LIN {X 0,Y 265.309,Z 598.013,A -85,B 0,C 180,E1 -22713.344,E2 -22713.344} C_VEL
LIN {X 0,Y 272.116,Z 583.48,A -85,B 0,C 180,E1 -22714.4,E2 -22714.4} C_VEL
LIN {X 0,Y 277.319,Z 569.981,A -85,B 0,C 180,E1 -22715.135,E2 -22715.135} C_VEL
LIN {X 0,Y 276.814,Z 571.467,A -85,B 0,C 180,E1 -22715.465,E2 -22715.465} C_VEL
LIN {X 0,Y 273.942,Z 579.172,A -85,B 0,C 180,E1 -22715.833,E2 -22715.833} C_VEL
LIN {X 0,Y 271.697,Z 584.628,A -85,B 0,C 180,E1 -22715.976,E2 -22715.976} C_VEL
LIN {X 0,Y 263.827,Z 600.629,A -85,B 0,C 180,E1 -22715.795,E2 -22715.795} C_VEL
LIN {X 0,Y 261.002,Z 605.716,A -85,B 0,C 180,E1 -22715.928,E2 -22715.928} C_VEL
LIN {X 0,Y 260.072,Z 607.334,A -85,B 0,C 180,E1 -22716.034,E2 -22716.034} C_VEL
LIN {X 0,Y 251.746,Z 620.764,A -85,B 0,C 180,E1 -22717.282,E2 -22717.282} C_VEL
LIN {X 0,Y 243.261,Z 632.852,A -85,B 0,C 180,E1 -22718.732,E2 -22718.732} C_VEL
LIN {X 0,Y 233.8,Z 644.794,A -85,B 0,C 180,E1 -22720.62,E2 -22720.62} C_VEL
LIN {X 0,Y 224.848,Z 655.062,A -85,B 0,C 180,E1 -22722.729,E2 -22722.729} C_VEL
LIN {X 0,Y 215.182,Z 665.04,A -85,B 0,C 180,E1 -22725.393,E2 -22725.393} C_VEL
LIN {X 0,Y 206.221,Z 673.491,A -85,B 0,C 180,E1 -22728.348,E2 -22728.348} C_VEL
LIN {X 0,Y 198.032,Z 680.601,A -85,B 0,C 180,E1 -22731.603,E2 -22731.603} C_VEL
LIN {X 0,Y 190.807,Z 686.435,A -85,B 0,C 180,E1 -22735.183,E2 -22735.183} C_VEL
LIN {X 0,Y 183.186,Z 692.152,A -85,B 0,C 180,E1 -22740.079,E2 -22740.079} C_VEL
LIN {X 0,Y 178.076,Z 695.522,A -85,B 0,C 180,E1 -22744.267,E2 -22744.267} C_VEL
LIN {X 0,Y 174.051,Z 697.841,A -85,B 0,C 180,E1 -22748.687,E2 -22748.687} C_VEL
LIN {X 0,Y 171.345,Z 699.174,A -85,B 0,C 180,E1 -22753.311,E2 -22753.311} C_VEL
LIN {X 0,Y 169.67,Z 699.443,A -85,B 0,C 180,E1 -22758.044,E2 -22758.044} C_VEL
LIN {X 0,Y 168.987,Z 698.624,A -85,B 0,C 180,E1 -22762.829,E2 -22762.829} C_VEL
LIN {X 0,Y 169.136,Z 696.706,A -85,B 0,C 180,E1 -22767.615,E2 -22767.615} C_VEL
LIN {X 0,Y 169.279,Z 695.29,A -85,B 0,C 180,E1 -22769.996,E2 -22769.996} C_VEL
LIN {X 0,Y 169.245,Z 692.646,A -85,B 0,C 180,E1 -22773.352,E2 -22773.352} C_VEL
LIN {X 0,Y 169.28,Z 688.807,A -85,B 0,C 180,E1 -22777.151,E2 -22777.151} C_VEL
LIN {X 0,Y 169.775,Z 682.485,A -85,B 0,C 180,E1 -22781.942,E2 -22781.942} C_VEL
LIN {X 0,Y 170.866,Z 675.519,A -85,B 0,C 180,E1 -22786.115,E2 -22786.115} C_VEL
LIN {X 0,Y 172.718,Z 666.779,A -85,B 0,C 180,E1 -22790.36,E2 -22790.36} C_VEL
LIN {X 0,Y 175.16,Z 656.817,A -85,B 0,C 180,E1 -22794.28,E2 -22794.28} C_VEL
LIN {X 0,Y 177.808,Z 646.284,A -85,B 0,C 180,E1 -22797.669,E2 -22797.669} C_VEL
LIN {X 0,Y 180.909,Z 634.538,A -85,B 0,C 180,E1 -22800.765,E2 -22800.765} C_VEL
LIN {X 0,Y 184.216,Z 621.341,A -85,B 0,C 180,E1 -22803.582,E2 -22803.582} C_VEL
LIN {X 0,Y 187.346,Z 607.954,A -85,B 0,C 180,E1 -22805.88,E2 -22805.88} C_VEL
LIN {X 0,Y 190.597,Z 592.477,A -85,B 0,C 180,E1 -22807.971,E2 -22807.971} C_VEL
LIN {X 0,Y 193.235,Z 577.622,A -85,B 0,C 180,E1 -22809.525,E2 -22809.525} C_VEL
LIN {X 0,Y 195.597,Z 561.354,A -85,B 0,C 180,E1 -22810.781,E2 -22810.781} C_VEL
LIN {X 0,Y 197.639,Z 540.646,A -85,B 0,C 180,E1 -22811.89,E2 -22811.89} C_VEL
LIN {X 0,Y 204.347,Z 466.811,A -85,B 0,C 180,E1 -22815.376,E2 -22815.376} C_VEL
LIN {X 0,Y 196.162,Z 445.438,A -85,B 0,C 180,E1 -22818.116,E2 -22818.116} C_VEL
LIN {X 0,Y 186.895,Z 423.814,A -85,B 0,C 180,E1 -22821.346,E2 -22821.346} C_VEL
LIN {X 0,Y 180.833,Z 410.824,A -85,B 0,C 180,E1 -22823.629,E2 -22823.629} C_VEL
LIN {X 0,Y 174.86,Z 400.671,A -85,B 0,C 180,E1 -22825.813,E2 -22825.813} C_VEL
LIN {X 0,Y 172.955,Z 397.334,A -85,B 0,C 180,E1 -22826.558,E2 -22826.558} C_VEL
LIN {X 0,Y 171.581,Z 394.658,A -85,B 0,C 180,E1 -22827.132,E2 -22827.132} C_VEL
LIN {X 0,Y 171.407,Z 393.76,A -85,B 0,C 180,E1 -22827.269,E2 -22827.269} C_VEL
LIN {X 0,Y 171.396,Z 393.759,A -85,B 0,C 180,E1 -22830.525,E2 -22830.525} C_VEL
LIN {X 0,Y 171.391,Z 393.755,A -85,B 0,C 180,E1 -22835.792,E2 -22835.792} C_VEL
LIN {X 0,Y 171.496,Z 393.731,A -85,B 0,C 180,E1 -22840.863,E2 -22840.863} C_VEL
LIN {X 0,Y 171.535,Z 393.744,A -85,B 0,C 180,E1 -22845.77,E2 -22845.77} C_VEL
LIN {X 0,Y 171.829,Z 393.686,A -85,B 0,C 180,E1 -22850.584,E2 -22850.584} C_VEL
LIN {X 0,Y 171.769,Z 393.713,A -85,B 0,C 180,E1 -22855.307,E2 -22855.307} C_VEL
LIN {X 0,Y 172.297,Z 393.65,A -85,B 0,C 180,E1 -22860.001,E2 -22860.001} C_VEL
LIN {X 0,Y 171.83,Z 393.704,A -85,B 0,C 180,E1 -22866.865,E2 -22866.865} C_VEL
LIN {X 0,Y 171.755,Z 393.708,A -85,B 0,C 180,E1 -22870.895,E2 -22870.895} C_VEL
LIN {X 0,Y 171.498,Z 393.739,A -85,B 0,C 180,E1 -22876.671,E2 -22876.671} C_VEL
LIN {X 0,Y 171.468,Z 393.746,A -85,B 0,C 180,E1 -22879.502,E2 -22879.502} C_VEL
LIN {X 0,Y 171.392,Z 393.749,A -85,B 0,C 180,E1 -22885.572,E2 -22885.572} C_VEL
LIN {X 0,Y 171.408,Z 393.757,A -85,B 0,C 180,E1 -22890.575,E2 -22890.575} C_VEL
LIN {X 0,Y 171.383,Z 393.751,A -85,B 0,C 180,E1 -22895.038,E2 -22895.038} C_VEL
LIN {X 0,Y 171.335,Z 393.766,A -85,B 0,C 180,E1 -22898.804,E2 -22898.804} C_VEL
LIN {X 0,Y 171.311,Z 393.764,A -85,B 0,C 180,E1 -22904.222,E2 -22904.222} C_VEL
LIN {X 0,Y 171.323,Z 393.764,A -85,B 0,C 180,E1 -22908.983,E2 -22908.983} C_VEL
LIN {X 0,Y 171.354,Z 393.757,A -85,B 0,C 180,E1 -22912.037,E2 -22912.037} C_VEL
LIN {X 0,Y 171.393,Z 393.76,A -85,B 0,C 180,E1 -22915.097,E2 -22915.097} C_VEL
LIN {X 0,Y 171.404,Z 393.757,A -85,B 0,C 180,E1 -22920.53,E2 -22920.53} C_VEL
LIN {X 0,Y 171.427,Z 393.749,A -85,B 0,C 180,E1 -22925.801,E2 -22925.801} C_VEL
LIN {X 0,Y 171.517,Z 393.743,A -85,B 0,C 180,E1 -22930.868,E2 -22930.868} C_VEL
LIN {X 0,Y 171.561,Z 393.709,A -85,B 0,C 180,E1 -22935.775,E2 -22935.775} C_VEL
LIN {X 0,Y 171.844,Z 393.704,A -85,B 0,C 180,E1 -22940.588,E2 -22940.588} C_VEL
LIN {X 0,Y 171.784,Z 393.691,A -85,B 0,C 180,E1 -22945.31,E2 -22945.31} C_VEL
LIN {X 0,Y 172.313,Z 393.647,A -85,B 0,C 180,E1 -22950.003,E2 -22950.003} C_VEL
LIN {X 0,Y 171.79,Z 393.709,A -85,B 0,C 180,E1 -22954.697,E2 -22954.697} C_VEL
LIN {X 0,Y 171.848,Z 393.694,A -85,B 0,C 180,E1 -22959.419,E2 -22959.419} C_VEL
LIN {X 0,Y 171.547,Z 393.732,A -85,B 0,C 180,E1 -22964.612,E2 -22964.612} C_VEL
LIN {X 0,Y 172.401,Z 396.369,A -85,B 0,C 180,E1 -22965.066,E2 -22965.066} C_VEL
LIN {X 0,Y 174.007,Z 398.835,A -85,B 0,C 180,E1 -22965.674,E2 -22965.674} C_VEL
LIN {X 0,Y 180.352,Z 409.954,A -85,B 0,C 180,E1 -22968.021,E2 -22968.021} C_VEL
LIN {X 0,Y 190.153,Z 428.23,A -85,B 0,C 180,E1 -22971.426,E2 -22971.426} C_VEL
LIN {X 0,Y 199.911,Z 448.405,A -85,B 0,C 180,E1 -22974.543,E2 -22974.543} C_VEL
LIN {X 0,Y 204.128,Z 458.127,A -85,B 0,C 180,E1 -22975.853,E2 -22975.853} C_VEL
LIN {X 0,Y 204.377,Z 459.114,A -85,B 0,C 180,E1 -22975.953,E2 -22975.953} C_VEL
LIN {X 0,Y 196.155,Z 546.834,A -85,B 0,C 180,E1 -22980.109,E2 -22980.109} C_VEL
LIN {X 0,Y 194.151,Z 562.34,A -85,B 0,C 180,E1 -22981.218,E2 -22981.218} C_VEL
LIN {X 0,Y 191.648,Z 578.197,A -85,B 0,C 180,E1 -22982.776,E2 -22982.776} C_VEL
LIN {X 0,Y 188.749,Z 592.941,A -85,B 0,C 180,E1 -22984.643,E2 -22984.643} C_VEL
LIN {X 0,Y 185.649,Z 607.015,A -85,B 0,C 180,E1 -22986.896,E2 -22986.896} C_VEL
LIN {X 0,Y 182.391,Z 620.466,A -85,B 0,C 180,E1 -22989.586,E2 -22989.586} C_VEL
LIN {X 0,Y 179.209,Z 632.933,A -85,B 0,C 180,E1 -22992.665,E2 -22992.665} C_VEL
LIN {X 0,Y 176.477,Z 643.375,A -85,B 0,C 180,E1 -22995.798,E2 -22995.798} C_VEL
LIN {X 0,Y 173.855,Z 654.051,A -85,B 0,C 180,E1 -22999.699,E2 -22999.699} C_VEL
LIN {X 0,Y 171.827,Z 662.83,A -85,B 0,C 180,E1 -23003.624,E2 -23003.624} C_VEL
LIN {X 0,Y 170.237,Z 671.195,A -85,B 0,C 180,E1 -23008.239,E2 -23008.239} C_VEL
LIN {X 0,Y 169.225,Z 677.779,A -85,B 0,C 180,E1 -23012.816,E2 -23012.816} C_VEL
LIN {X 0,Y 168.701,Z 681.95,A -85,B 0,C 180,E1 -23016.428,E2 -23016.428} C_VEL
LIN {X 0,Y 168.411,Z 685.58,A -85,B 0,C 180,E1 -23020.497,E2 -23020.497} C_VEL
LIN {X 0,Y 168.556,Z 687.74,A -85,B 0,C 180,E1 -23023.545,E2 -23023.545} C_VEL
LIN {X 0,Y 169.088,Z 689.995,A -85,B 0,C 180,E1 -23028.005,E2 -23028.005} C_VEL
LIN {X 0,Y 170.558,Z 691.354,A -85,B 0,C 180,E1 -23032.898,E2 -23032.898} C_VEL
LIN {X 0,Y 172.858,Z 691.573,A -85,B 0,C 180,E1 -23037.669,E2 -23037.669} C_VEL
LIN {X 0,Y 176.211,Z 690.641,A -85,B 0,C 180,E1 -23042.285,E2 -23042.285} C_VEL
LIN {X 0,Y 180.649,Z 688.635,A -85,B 0,C 180,E1 -23046.702,E2 -23046.702} C_VEL
LIN {X 0,Y 186.124,Z 685.561,A -85,B 0,C 180,E1 -23050.882,E2 -23050.882} C_VEL
LIN {X 0,Y 192.617,Z 681.32,A -85,B 0,C 180,E1 -23054.797,E2 -23054.797} C_VEL
LIN {X 0,Y 200.065,Z 675.862,A -85,B 0,C 180,E1 -23058.43,E2 -23058.43} C_VEL
LIN {X 0,Y 208.432,Z 669.025,A -85,B 0,C 180,E1 -23061.771,E2 -23061.771} C_VEL
LIN {X 0,Y 215.958,Z 662.271,A -85,B 0,C 180,E1 -23064.321,E2 -23064.321} C_VEL
LIN {X 0,Y 226.24,Z 652.056,A -85,B 0,C 180,E1 -23067.27,E2 -23067.27} C_VEL
LIN {X 0,Y 235.563,Z 641.593,A -85,B 0,C 180,E1 -23069.545,E2 -23069.545} C_VEL
LIN {X 0,Y 245.162,Z 629.6,A -85,B 0,C 180,E1 -23071.544,E2 -23071.544} C_VEL
LIN {X 0,Y 254.447,Z 616.272,A -85,B 0,C 180,E1 -23073.257,E2 -23073.257} C_VEL
LIN {X 0,Y 262.74,Z 602.507,A -85,B 0,C 180,E1 -23074.602,E2 -23074.602} C_VEL
LIN {X 0,Y 266.574,Z 595.227,A -85,B 0,C 180,E1 -23075.183,E2 -23075.183} C_VEL
LIN {X 0,Y 260.072,Z 607.334,A -85,B 0,C 180,E1 -23076.034,E2 -23076.034} C_VEL
LIN {X 0,Y 257.087,Z 612.343,A -85,B 0,C 180,E1 -23076.29,E2 -23076.29} C_VEL
LIN {X 0,Y 246.93,Z 626.983,A -85,B 0,C 180,E1 -23076.519,E2 -23076.519} C_VEL
LIN {X 0,Y 243.455,Z 631.505,A -85,B 0,C 180,E1 -23076.819,E2 -23076.819} C_VEL
LIN {X 0,Y 242.341,Z 632.921,A -85,B 0,C 180,E1 -23076.983,E2 -23076.983} C_VEL
LIN {X 0,Y 232.271,Z 645.047,A -85,B 0,C 180,E1 -23078.815,E2 -23078.815} C_VEL
LIN {X 0,Y 222.913,Z 655.104,A -85,B 0,C 180,E1 -23080.825,E2 -23080.825} C_VEL
LIN {X 0,Y 212.809,Z 664.976,A -85,B 0,C 180,E1 -23083.399,E2 -23083.399} C_VEL
LIN {X 0,Y 203.374,Z 673.297,A -85,B 0,C 180,E1 -23086.276,E2 -23086.276} C_VEL
LIN {X 0,Y 194.708,Z 680.311,A -85,B 0,C 180,E1 -23089.477,E2 -23089.477} C_VEL
LIN {X 0,Y 186.796,Z 686.155,A -85,B 0,C 180,E1 -23092.985,E2 -23092.985} C_VEL
LIN {X 0,Y 180.082,Z 690.756,A -85,B 0,C 180,E1 -23096.878,E2 -23096.878} C_VEL
LIN {X 0,Y 174.271,Z 694.399,A -85,B 0,C 180,E1 -23101.054,E2 -23101.054} C_VEL
LIN {X 0,Y 169.355,Z 697.037,A -85,B 0,C 180,E1 -23105.478,E2 -23105.478} C_VEL
LIN {X 0,Y 165.814,Z 698.599,A -85,B 0,C 180,E1 -23110.176,E2 -23110.176} C_VEL
LIN {X 0,Y 163.412,Z 699.182,A -85,B 0,C 180,E1 -23115.042,E2 -23115.042} C_VEL
LIN {X 0,Y 162.216,Z 698.761,A -85,B 0,C 180,E1 -23120.017,E2 -23120.017} C_VEL
LIN {X 0,Y 161.906,Z 697.196,A -85,B 0,C 180,E1 -23125.016,E2 -23125.016} C_VEL
LIN {X 0,Y 162.081,Z 695.984,A -85,B 0,C 180,E1 -23127.511,E2 -23127.511} C_VEL
LIN {X 0,Y 162.222,Z 694.453,A -85,B 0,C 180,E1 -23129.996,E2 -23129.996} C_VEL
LIN {X 0,Y 162.204,Z 691.823,A -85,B 0,C 180,E1 -23133.347,E2 -23133.347} C_VEL
LIN {X 0,Y 162.256,Z 687.647,A -85,B 0,C 180,E1 -23137.462,E2 -23137.462} C_VEL
LIN {X 0,Y 162.595,Z 682.924,A -85,B 0,C 180,E1 -23141.212,E2 -23141.212} C_VEL
LIN {X 0,Y 163.809,Z 675.047,A -85,B 0,C 180,E1 -23146.189,E2 -23146.189} C_VEL
LIN {X 0,Y 165.581,Z 666.653,A -85,B 0,C 180,E1 -23150.421,E2 -23150.421} C_VEL
LIN {X 0,Y 168.212,Z 656.197,A -85,B 0,C 180,E1 -23154.692,E2 -23154.692} C_VEL
LIN {X 0,Y 170.935,Z 645.589,A -85,B 0,C 180,E1 -23158.213,E2 -23158.213} C_VEL
LIN {X 0,Y 174.342,Z 632.997,A -85,B 0,C 180,E1 -23161.6,E2 -23161.6} C_VEL
LIN {X 0,Y 177.572,Z 620.489,A -85,B 0,C 180,E1 -23164.328,E2 -23164.328} C_VEL
LIN {X 0,Y 180.782,Z 607.031,A -85,B 0,C 180,E1 -23166.702,E2 -23166.702} C_VEL
LIN {X 0,Y 184.15,Z 591.506,A -85,B 0,C 180,E1 -23168.849,E2 -23168.849} C_VEL
LIN {X 0,Y 187.11,Z 575.285,A -85,B 0,C 180,E1 -23170.557,E2 -23170.557} C_VEL
LIN {X 0,Y 189.456,Z 559.085,A -85,B 0,C 180,E1 -23171.798,E2 -23171.798} C_VEL
LIN {X 0,Y 192.546,Z 526.859,A -85,B 0,C 180,E1 -23173.48,E2 -23173.48} C_VEL
LIN {X 0,Y 198.059,Z 468.566,A -85,B 0,C 180,E1 -23176.293,E2 -23176.293} C_VEL
LIN {X 0,Y 190.091,Z 447.695,A -85,B 0,C 180,E1 -23179.074,E2 -23179.074} C_VEL
LIN {X 0,Y 180.267,Z 424.517,A -85,B 0,C 180,E1 -23182.73,E2 -23182.73} C_VEL
LIN {X 0,Y 174.823,Z 413.322,A -85,B 0,C 180,E1 -23184.82,E2 -23184.82} C_VEL
LIN {X 0,Y 167.745,Z 401.33,A -85,B 0,C 180,E1 -23187.598,E2 -23187.598} C_VEL
LIN {X 0,Y 166.305,Z 398.723,A -85,B 0,C 180,E1 -23188.218,E2 -23188.218} C_VEL
LIN {X 0,Y 164.725,Z 396.211,A -85,B 0,C 180,E1 -23188.875,E2 -23188.875} C_VEL
LIN {X 0,Y 164.37,Z 394.637,A -85,B 0,C 180,E1 -23189.131,E2 -23189.131} C_VEL
LIN {X 0,Y 164.345,Z 394.626,A -85,B 0,C 180,E1 -23194.683,E2 -23194.683} C_VEL
LIN {X 0,Y 164.404,Z 394.617,A -85,B 0,C 180,E1 -23200.117,E2 -23200.117} C_VEL
LIN {X 0,Y 164.464,Z 394.625,A -85,B 0,C 180,E1 -23205.144,E2 -23205.144} C_VEL
LIN {X 0,Y 164.75,Z 394.565,A -85,B 0,C 180,E1 -23210.176,E2 -23210.176} C_VEL
LIN {X 0,Y 164.805,Z 394.576,A -85,B 0,C 180,E1 -23212.651,E2 -23212.651} C_VEL
LIN {X 0,Y 165.261,Z 394.526,A -85,B 0,C 180,E1 -23220.001,E2 -23220.001} C_VEL
LIN {X 0,Y 164.808,Z 394.581,A -85,B 0,C 180,E1 -23227.351,E2 -23227.351} C_VEL
LIN {X 0,Y 164.69,Z 394.588,A -85,B 0,C 180,E1 -23231.059,E2 -23231.059} C_VEL
LIN {X 0,Y 164.42,Z 394.618,A -85,B 0,C 180,E1 -23237.411,E2 -23237.411} C_VEL
LIN {X 0,Y 164.409,Z 394.628,A -85,B 0,C 180,E1 -23239.998,E2 -23239.998} C_VEL
LIN {X 0,Y 164.328,Z 394.628,A -85,B 0,C 180,E1 -23246.097,E2 -23246.097} C_VEL
LIN {X 0,Y 164.348,Z 394.637,A -85,B 0,C 180,E1 -23251.22,E2 -23251.22} C_VEL
LIN {X 0,Y 164.271,Z 394.644,A -85,B 0,C 180,E1 -23256.796,E2 -23256.796} C_VEL
LIN {X 0,Y 164.278,Z 394.643,A -85,B 0,C 180,E1 -23259.921,E2 -23259.921} C_VEL
LIN {X 0,Y 164.273,Z 394.635,A -85,B 0,C 180,E1 -23263.345,E2 -23263.345} C_VEL
LIN {X 0,Y 164.253,Z 394.648,A -85,B 0,C 180,E1 -23266.801,E2 -23266.801} C_VEL
LIN {X 0,Y 164.283,Z 394.633,A -85,B 0,C 180,E1 -23270.359,E2 -23270.359} C_VEL
LIN {X 0,Y 164.32,Z 394.641,A -85,B 0,C 180,E1 -23274.355,E2 -23274.355} C_VEL
LIN {X 0,Y 164.363,Z 394.626,A -85,B 0,C 180,E1 -23279.134,E2 -23279.134} C_VEL
LIN {X 0,Y 164.384,Z 394.628,A -85,B 0,C 180,E1 -23284.693,E2 -23284.693} C_VEL
LIN {X 0,Y 164.418,Z 394.628,A -85,B 0,C 180,E1 -23290.118,E2 -23290.118} C_VEL
LIN {X 0,Y 164.489,Z 394.587,A -85,B 0,C 180,E1 -23295.15,E2 -23295.15} C_VEL
LIN {X 0,Y 164.766,Z 394.587,A -85,B 0,C 180,E1 -23300.18,E2 -23300.18} C_VEL
LIN {X 0,Y 164.821,Z 394.571,A -85,B 0,C 180,E1 -23302.654,E2 -23302.654} C_VEL
LIN {X 0,Y 165.277,Z 394.523,A -85,B 0,C 180,E1 -23310.004,E2 -23310.004} C_VEL
LIN {X 0,Y 164.825,Z 394.578,A -85,B 0,C 180,E1 -23317.353,E2 -23317.353} C_VEL
LIN {X 0,Y 164.701,Z 394.593,A -85,B 0,C 180,E1 -23321.053,E2 -23321.053} C_VEL
LIN {X 0,Y 164.572,Z 394.731,A -85,B 0,C 180,E1 -23322.802,E2 -23322.802} C_VEL
LIN {X 0,Y 165.635,Z 397.611,A -85,B 0,C 180,E1 -23323.342,E2 -23323.342} C_VEL
LIN {X 0,Y 167.007,Z 399.607,A -85,B 0,C 180,E1 -23323.894,E2 -23323.894} C_VEL
LIN {X 0,Y 174.83,Z 413.347,A -85,B 0,C 180,E1 -23327.015,E2 -23327.015} C_VEL
LIN {X 0,Y 183.507,Z 429.583,A -85,B 0,C 180,E1 -23330.166,E2 -23330.166} C_VEL
LIN {X 0,Y 194.197,Z 451.552,A -85,B 0,C 180,E1 -23333.729,E2 -23333.729} C_VEL
LIN {X 0,Y 198.049,Z 460.512,A -85,B 0,C 180,E1 -23334.984,E2 -23334.984} C_VEL
LIN {X 0,Y 189.736,Z 546.86,A -85,B 0,C 180,E1 -23339.216,E2 -23339.216} C_VEL
LIN {X 0,Y 187.516,Z 563.366,A -85,B 0,C 180,E1 -23340.453,E2 -23340.453} C_VEL
LIN {X 0,Y 185.074,Z 578.251,A -85,B 0,C 180,E1 -23341.975,E2 -23341.975} C_VEL
LIN {X 0,Y 182.06,Z 593.007,A -85,B 0,C 180,E1 -23343.904,E2 -23343.904} C_VEL
LIN {X 0,Y 178.874,Z 607.033,A -85,B 0,C 180,E1 -23346.228,E2 -23346.228} C_VEL
LIN {X 0,Y 175.44,Z 620.856,A -85,B 0,C 180,E1 -23349.09,E2 -23349.09} C_VEL
LIN {X 0,Y 172.185,Z 633.307,A -85,B 0,C 180,E1 -23352.284,E2 -23352.284} C_VEL
LIN {X 0,Y 169.119,Z 644.742,A -85,B 0,C 180,E1 -23355.886,E2 -23355.886} C_VEL
LIN {X 0,Y 166.503,Z 655.245,A -85,B 0,C 180,E1 -23359.958,E2 -23359.958} C_VEL
LIN {X 0,Y 164.361,Z 664.416,A -85,B 0,C 180,E1 -23364.34,E2 -23364.34} C_VEL
LIN {X 0,Y 162.963,Z 671.977,A -85,B 0,C 180,E1 -23368.833,E2 -23368.833} C_VEL
LIN {X 0,Y 162.111,Z 677.559,A -85,B 0,C 180,E1 -23372.921,E2 -23372.921} C_VEL
LIN {X 0,Y 161.542,Z 682.055,A -85,B 0,C 180,E1 -23376.948,E2 -23376.948} C_VEL
LIN {X 0,Y 161.331,Z 685.518,A -85,B 0,C 180,E1 -23380.929,E2 -23380.929} C_VEL
LIN {X 0,Y 161.541,Z 688.197,A -85,B 0,C 180,E1 -23384.868,E2 -23384.868} C_VEL
LIN {X 0,Y 162.42,Z 690.538,A -85,B 0,C 180,E1 -23390.032,E2 -23390.032} C_VEL
LIN {X 0,Y 164.313,Z 691.706,A -85,B 0,C 180,E1 -23395.092,E2 -23395.092} C_VEL
LIN {X 0,Y 167.11,Z 691.771,A -85,B 0,C 180,E1 -23399.999,E2 -23399.999} C_VEL
LIN {X 0,Y 171.078,Z 690.75,A -85,B 0,C 180,E1 -23404.712,E2 -23404.712} C_VEL
LIN {X 0,Y 176.153,Z 688.62,A -85,B 0,C 180,E1 -23409.182,E2 -23409.182} C_VEL
LIN {X 0,Y 182.257,Z 685.406,A -85,B 0,C 180,E1 -23413.377,E2 -23413.377} C_VEL
LIN {X 0,Y 189.395,Z 681.103,A -85,B 0,C 180,E1 -23417.269,E2 -23417.269} C_VEL
LIN {X 0,Y 197.541,Z 675.543,A -85,B 0,C 180,E1 -23420.84,E2 -23420.84} C_VEL
LIN {X 0,Y 206.495,Z 668.649,A -85,B 0,C 180,E1 -23424.105,E2 -23424.105} C_VEL
LIN {X 0,Y 216.315,Z 660.244,A -85,B 0,C 180,E1 -23427.055,E2 -23427.055} C_VEL
LIN {X 0,Y 226.267,Z 650.649,A -85,B 0,C 180,E1 -23429.572,E2 -23429.572} C_VEL
LIN {X 0,Y 235.14,Z 641.085,A -85,B 0,C 180,E1 -23431.537,E2 -23431.537} C_VEL
LIN {X 0,Y 246.03,Z 627.844,A -85,B 0,C 180,E1 -23433.601,E2 -23433.601} C_VEL
LIN {X 0,Y 253.972,Z 616.755,A -85,B 0,C 180,E1 -23434.918,E2 -23434.918} C_VEL
LIN {X 0,Y 253.57,Z 617.352,A -85,B 0,C 180,E1 -23435.252,E2 -23435.252} C_VEL
LIN {X 0,Y 244.958,Z 629.559,A -85,B 0,C 180,E1 -23436.547,E2 -23436.547} C_VEL
LIN {X 0,Y 242.341,Z 632.921,A -85,B 0,C 180,E1 -23436.983,E2 -23436.983} C_VEL
LIN {X 0,Y 238.762,Z 637.308,A -85,B 0,C 180,E1 -23437.415,E2 -23437.415} C_VEL
LIN {X 0,Y 226.667,Z 650.086,A -85,B 0,C 180,E1 -23438.136,E2 -23438.136} C_VEL
LIN {X 0,Y 222.719,Z 653.943,A -85,B 0,C 180,E1 -23438.631,E2 -23438.631} C_VEL
LIN {X 0,Y 221.493,Z 655.128,A -85,B 0,C 180,E1 -23438.867,E2 -23438.867} C_VEL
LIN {X 0,Y 210.73,Z 664.996,A -85,B 0,C 180,E1 -23441.372,E2 -23441.372} C_VEL
LIN {X 0,Y 200.849,Z 673.215,A -85,B 0,C 180,E1 -23444.162,E2 -23444.162} C_VEL
LIN {X 0,Y 192.191,Z 679.736,A -85,B 0,C 180,E1 -23447.063,E2 -23447.063} C_VEL
LIN {X 0,Y 183.25,Z 685.885,A -85,B 0,C 180,E1 -23450.739,E2 -23450.739} C_VEL
LIN {X 0,Y 174.205,Z 691.497,A -85,B 0,C 180,E1 -23455.608,E2 -23455.608} C_VEL
LIN {X 0,Y 168.087,Z 694.815,A -85,B 0,C 180,E1 -23459.881,E2 -23459.881} C_VEL
LIN {X 0,Y 162.899,Z 697.166,A -85,B 0,C 180,E1 -23464.438,E2 -23464.438} C_VEL
LIN {X 0,Y 159.102,Z 698.562,A -85,B 0,C 180,E1 -23469.302,E2 -23469.302} C_VEL
LIN {X 0,Y 156.513,Z 698.895,A -85,B 0,C 180,E1 -23474.366,E2 -23474.366} C_VEL
LIN {X 0,Y 155.193,Z 698.241,A -85,B 0,C 180,E1 -23479.56,E2 -23479.56} C_VEL
LIN {X 0,Y 154.844,Z 696.538,A -85,B 0,C 180,E1 -23484.788,E2 -23484.788} C_VEL
LIN {X 0,Y 155.031,Z 695.248,A -85,B 0,C 180,E1 -23487.398,E2 -23487.398} C_VEL
LIN {X 0,Y 155.143,Z 692.648,A -85,B 0,C 180,E1 -23491.294,E2 -23491.294} C_VEL
LIN {X 0,Y 155.156,Z 689.213,A -85,B 0,C 180,E1 -23495.194,E2 -23495.194} C_VEL
LIN {X 0,Y 155.44,Z 683.237,A -85,B 0,C 180,E1 -23500.415,E2 -23500.415} C_VEL
LIN {X 0,Y 156.531,Z 675.556,A -85,B 0,C 180,E1 -23505.624,E2 -23505.624} C_VEL
LIN {X 0,Y 158.267,Z 667.228,A -85,B 0,C 180,E1 -23510.125,E2 -23510.125} C_VEL
LIN {X 0,Y 160.842,Z 657.16,A -85,B 0,C 180,E1 -23514.521,E2 -23514.521} C_VEL
LIN {X 0,Y 163.589,Z 646.763,A -85,B 0,C 180,E1 -23518.197,E2 -23518.197} C_VEL
LIN {X 0,Y 166.98,Z 634.461,A -85,B 0,C 180,E1 -23521.738,E2 -23521.738} C_VEL
LIN {X 0,Y 170.463,Z 621.478,A -85,B 0,C 180,E1 -23524.744,E2 -23524.744} C_VEL
LIN {X 0,Y 173.888,Z 607.625,A -85,B 0,C 180,E1 -23527.314,E2 -23527.314} C_VEL
LIN {X 0,Y 177.348,Z 592.313,A -85,B 0,C 180,E1 -23529.529,E2 -23529.529} C_VEL
LIN {X 0,Y 180.354,Z 576.352,A -85,B 0,C 180,E1 -23531.296,E2 -23531.296} C_VEL
LIN {X 0,Y 182.892,Z 559.849,A -85,B 0,C 180,E1 -23532.626,E2 -23532.626} C_VEL
LIN {X 0,Y 185.341,Z 535.37,A -85,B 0,C 180,E1 -23534.001,E2 -23534.001} C_VEL
LIN {X 0,Y 191.807,Z 470.279,A -85,B 0,C 180,E1 -23537.265,E2 -23537.265} C_VEL
LIN {X 0,Y 184.193,Z 450.466,A -85,B 0,C 180,E1 -23540.009,E2 -23540.009} C_VEL
LIN {X 0,Y 175.101,Z 428.62,A -85,B 0,C 180,E1 -23543.572,E2 -23543.572} C_VEL
LIN {X 0,Y 169.951,Z 417.871,A -85,B 0,C 180,E1 -23545.64,E2 -23545.64} C_VEL
LIN {X 0,Y 161.646,Z 403.553,A -85,B 0,C 180,E1 -23549.098,E2 -23549.098} C_VEL
LIN {X 0,Y 159.095,Z 399.449,A -85,B 0,C 180,E1 -23550.201,E2 -23550.201} C_VEL
LIN {X 0,Y 157.53,Z 396.844,A -85,B 0,C 180,E1 -23550.913,E2 -23550.913} C_VEL
LIN {X 0,Y 157.248,Z 395.523,A -85,B 0,C 180,E1 -23551.158,E2 -23551.158} C_VEL
LIN {X 0,Y 157.254,Z 395.519,A -85,B 0,C 180,E1 -23556.283,E2 -23556.283} C_VEL
LIN {X 0,Y 157.347,Z 395.498,A -85,B 0,C 180,E1 -23559.702,E2 -23559.702} C_VEL
LIN {X 0,Y 157.397,Z 395.506,A -85,B 0,C 180,E1 -23564.461,E2 -23564.461} C_VEL
LIN {X 0,Y 157.673,Z 395.444,A -85,B 0,C 180,E1 -23569.73,E2 -23569.73} C_VEL
LIN {X 0,Y 157.744,Z 395.452,A -85,B 0,C 180,E1 -23572.32,E2 -23572.32} C_VEL
LIN {X 0,Y 158.223,Z 395.403,A -85,B 0,C 180,E1 -23580.001,E2 -23580.001} C_VEL
LIN {X 0,Y 157.746,Z 395.46,A -85,B 0,C 180,E1 -23587.682,E2 -23587.682} C_VEL
LIN {X 0,Y 157.619,Z 395.469,A -85,B 0,C 180,E1 -23591.225,E2 -23591.225} C_VEL
LIN {X 0,Y 157.398,Z 395.5,A -85,B 0,C 180,E1 -23595.541,E2 -23595.541} C_VEL
LIN {X 0,Y 157.293,Z 395.516,A -85,B 0,C 180,E1 -23600.944,E2 -23600.944} C_VEL
LIN {X 0,Y 157.256,Z 395.511,A -85,B 0,C 180,E1 -23606.652,E2 -23606.652} C_VEL
LIN {X 0,Y 157.258,Z 395.513,A -85,B 0,C 180,E1 -23612.432,E2 -23612.432} C_VEL
LIN {X 0,Y 157.25,Z 395.518,A -85,B 0,C 180,E1 -23616.447,E2 -23616.447} C_VEL
LIN {X 0,Y 157.182,Z 395.516,A -85,B 0,C 180,E1 -23622.121,E2 -23622.121} C_VEL
LIN {X 0,Y 157.183,Z 395.528,A -85,B 0,C 180,E1 -23627.886,E2 -23627.886} C_VEL
LIN {X 0,Y 157.253,Z 395.52,A -85,B 0,C 180,E1 -23633.56,E2 -23633.56} C_VEL
LIN {X 0,Y 157.275,Z 395.508,A -85,B 0,C 180,E1 -23638.108,E2 -23638.108} C_VEL
LIN {X 0,Y 157.306,Z 395.514,A -85,B 0,C 180,E1 -23643.468,E2 -23643.468} C_VEL
LIN {X 0,Y 157.36,Z 395.509,A -85,B 0,C 180,E1 -23649.704,E2 -23649.704} C_VEL
LIN {X 0,Y 157.421,Z 395.467,A -85,B 0,C 180,E1 -23654.467,E2 -23654.467} C_VEL
LIN {X 0,Y 157.688,Z 395.468,A -85,B 0,C 180,E1 -23659.735,E2 -23659.735} C_VEL
LIN {X 0,Y 157.759,Z 395.453,A -85,B 0,C 180,E1 -23662.324,E2 -23662.324} C_VEL
LIN {X 0,Y 158.24,Z 395.4,A -85,B 0,C 180,E1 -23670.004,E2 -23670.004} C_VEL
LIN {X 0,Y 157.763,Z 395.455,A -85,B 0,C 180,E1 -23677.684,E2 -23677.684} C_VEL
LIN {X 0,Y 157.689,Z 395.584,A -85,B 0,C 180,E1 -23680.871,E2 -23680.871} C_VEL
LIN {X 0,Y 158.632,Z 398.311,A -85,B 0,C 180,E1 -23681.412,E2 -23681.412} C_VEL
LIN {X 0,Y 160.15,Z 400.763,A -85,B 0,C 180,E1 -23682.084,E2 -23682.084} C_VEL
LIN {X 0,Y 168.215,Z 414.667,A -85,B 0,C 180,E1 -23685.485,E2 -23685.485} C_VEL
LIN {X 0,Y 176.846,Z 430.82,A -85,B 0,C 180,E1 -23688.814,E2 -23688.814} C_VEL
LIN {X 0,Y 185.269,Z 447.999,A -85,B 0,C 180,E1 -23691.837,E2 -23691.837} C_VEL
LIN {X 0,Y 191.764,Z 462.177,A -85,B 0,C 180,E1 -23694.003,E2 -23694.003} C_VEL
LIN {X 0,Y 183.257,Z 547.205,A -85,B 0,C 180,E1 -23698.324,E2 -23698.324} C_VEL
LIN {X 0,Y 180.917,Z 564.042,A -85,B 0,C 180,E1 -23699.633,E2 -23699.633} C_VEL
LIN {X 0,Y 178.059,Z 580.471,A -85,B 0,C 180,E1 -23701.4,E2 -23701.4} C_VEL
LIN {X 0,Y 174.754,Z 596.036,A -85,B 0,C 180,E1 -23703.585,E2 -23703.585} C_VEL
LIN {X 0,Y 171.542,Z 609.511,A -85,B 0,C 180,E1 -23705.986,E2 -23705.986} C_VEL
LIN {X 0,Y 168.011,Z 623.108,A -85,B 0,C 180,E1 -23708.995,E2 -23708.995} C_VEL
LIN {X 0,Y 164.533,Z 635.938,A -85,B 0,C 180,E1 -23712.537,E2 -23712.537} C_VEL
LIN {X 0,Y 161.377,Z 647.629,A -85,B 0,C 180,E1 -23716.577,E2 -23716.577} C_VEL
LIN {X 0,Y 158.746,Z 657.704,A -85,B 0,C 180,E1 -23720.884,E2 -23720.884} C_VEL
LIN {X 0,Y 156.9,Z 665.915,A -85,B 0,C 180,E1 -23725.172,E2 -23725.172} C_VEL
LIN {X 0,Y 155.818,Z 671.947,A -85,B 0,C 180,E1 -23728.985,E2 -23728.985} C_VEL
LIN {X 0,Y 155.019,Z 677.331,A -85,B 0,C 180,E1 -23733.039,E2 -23733.039} C_VEL
LIN {X 0,Y 154.428,Z 681.878,A -85,B 0,C 180,E1 -23737.242,E2 -23737.242} C_VEL
LIN {X 0,Y 154.249,Z 685.419,A -85,B 0,C 180,E1 -23741.4,E2 -23741.4} C_VEL
LIN {X 0,Y 154.406,Z 687.327,A -85,B 0,C 180,E1 -23744.15,E2 -23744.15} C_VEL
LIN {X 0,Y 155.178,Z 690.14,A -85,B 0,C 180,E1 -23749.562,E2 -23749.562} C_VEL
LIN {X 0,Y 157.015,Z 691.703,A -85,B 0,C 180,E1 -23754.863,E2 -23754.863} C_VEL
LIN {X 0,Y 159.834,Z 692.14,A -85,B 0,C 180,E1 -23759.999,E2 -23759.999} C_VEL
LIN {X 0,Y 163.854,Z 691.532,A -85,B 0,C 180,E1 -23764.92,E2 -23764.92} C_VEL
LIN {X 0,Y 169.032,Z 689.884,A -85,B 0,C 180,E1 -23769.573,E2 -23769.573} C_VEL
LIN {X 0,Y 175.264,Z 687.126,A -85,B 0,C 180,E1 -23773.921,E2 -23773.921} C_VEL
LIN {X 0,Y 182.573,Z 683.259,A -85,B 0,C 180,E1 -23777.935,E2 -23777.935} C_VEL
LIN {X 0,Y 190.896,Z 678.27,A -85,B 0,C 180,E1 -23781.601,E2 -23781.601} C_VEL
LIN {X 0,Y 200.103,Z 671.985,A -85,B 0,C 180,E1 -23784.926,E2 -23784.926} C_VEL
LIN {X 0,Y 210.129,Z 664.269,A -85,B 0,C 180,E1 -23787.92,E2 -23787.92} C_VEL
LIN {X 0,Y 220.855,Z 654.973,A -85,B 0,C 180,E1 -23790.607,E2 -23790.607} C_VEL
LIN {X 0,Y 232.266,Z 643.68,A -85,B 0,C 180,E1 -23793,E2 -23793} C_VEL
LIN {X 0,Y 242.546,Z 632.074,A -85,B 0,C 180,E1 -23794.833,E2 -23794.833} C_VEL
LIN {X 0,Y 241.151,Z 633.824,A -85,B 0,C 180,E1 -23795.308,E2 -23795.308} C_VEL
LIN {X 0,Y 232.448,Z 643.864,A -85,B 0,C 180,E1 -23796.75,E2 -23796.75} C_VEL
LIN {X 0,Y 222.642,Z 653.995,A -85,B 0,C 180,E1 -23798.62,E2 -23798.62} C_VEL
LIN {X 0,Y 221.493,Z 655.128,A -85,B 0,C 180,E1 -23798.867,E2 -23798.867} C_VEL
LIN {X 0,Y 217.55,Z 658.797,A -85,B 0,C 180,E1 -23799.523,E2 -23799.523} C_VEL
LIN {X 0,Y 210.136,Z 664.816,A -85,B 0,C 180,E1 -23800.273,E2 -23800.273} C_VEL
LIN {X 0,Y 202.613,Z 670.365,A -85,B 0,C 180,E1 -23801.148,E2 -23801.148} C_VEL
LIN {X 0,Y 198.556,Z 673.248,A -85,B 0,C 180,E1 -23802.014,E2 -23802.014} C_VEL
LIN {X 0,Y 188.893,Z 680.038,A -85,B 0,C 180,E1 -23805.011,E2 -23805.011} C_VEL
LIN {X 0,Y 177.861,Z 686.91,A -85,B 0,C 180,E1 -23809.305,E2 -23809.305} C_VEL
LIN {X 0,Y 171.961,Z 690.236,A -85,B 0,C 180,E1 -23812.186,E2 -23812.186} C_VEL
LIN {X 0,Y 165.064,Z 693.784,A -85,B 0,C 180,E1 -23816.388,E2 -23816.388} C_VEL
LIN {X 0,Y 159.126,Z 696.389,A -85,B 0,C 180,E1 -23820.929,E2 -23820.929} C_VEL
LIN {X 0,Y 154.219,Z 697.97,A -85,B 0,C 180,E1 -23825.782,E2 -23825.782} C_VEL
LIN {X 0,Y 150.933,Z 698.624,A -85,B 0,C 180,E1 -23830.973,E2 -23830.973} C_VEL
LIN {X 0,Y 148.787,Z 698.278,A -85,B 0,C 180,E1 -23836.335,E2 -23836.335} C_VEL
LIN {X 0,Y 147.85,Z 696.875,A -85,B 0,C 180,E1 -23841.797,E2 -23841.797} C_VEL
LIN {X 0,Y 147.99,Z 694.389,A -85,B 0,C 180,E1 -23847.274,E2 -23847.274} C_VEL
LIN {X 0,Y 148.103,Z 691.648,A -85,B 0,C 180,E1 -23851.355,E2 -23851.355} C_VEL
LIN {X 0,Y 148.092,Z 688.103,A -85,B 0,C 180,E1 -23855.442,E2 -23855.442} C_VEL
LIN {X 0,Y 148.318,Z 683.55,A -85,B 0,C 180,E1 -23859.542,E2 -23859.542} C_VEL
LIN {X 0,Y 149.308,Z 676.013,A -85,B 0,C 180,E1 -23865,E2 -23865} C_VEL
LIN {X 0,Y 150.943,Z 667.827,A -85,B 0,C 180,E1 -23869.724,E2 -23869.724} C_VEL
LIN {X 0,Y 153.431,Z 657.931,A -85,B 0,C 180,E1 -23874.342,E2 -23874.342} C_VEL
LIN {X 0,Y 156.239,Z 647.804,A -85,B 0,C 180,E1 -23878.18,E2 -23878.18} C_VEL
LIN {X 0,Y 159.615,Z 635.785,A -85,B 0,C 180,E1 -23881.891,E2 -23881.891} C_VEL
LIN {X 0,Y 163.27,Z 622.707,A -85,B 0,C 180,E1 -23885.13,E2 -23885.13} C_VEL
LIN {X 0,Y 166.643,Z 609.727,A -85,B 0,C 180,E1 -23887.695,E2 -23887.695} C_VEL
LIN {X 0,Y 170.344,Z 594.08,A -85,B 0,C 180,E1 -23890.134,E2 -23890.134} C_VEL
LIN {X 0,Y 173.4,Z 578.732,A -85,B 0,C 180,E1 -23891.966,E2 -23891.966} C_VEL
LIN {X 0,Y 176.096,Z 562.237,A -85,B 0,C 180,E1 -23893.404,E2 -23893.404} C_VEL
LIN {X 0,Y 178.151,Z 543.789,A -85,B 0,C 180,E1 -23894.539,E2 -23894.539} C_VEL
LIN {X 0,Y 185.451,Z 471.895,A -85,B 0,C 180,E1 -23898.271,E2 -23898.271} C_VEL
LIN {X 0,Y 178.203,Z 452.791,A -85,B 0,C 180,E1 -23901.073,E2 -23901.073} C_VEL
LIN {X 0,Y 169.663,Z 432.156,A -85,B 0,C 180,E1 -23904.555,E2 -23904.555} C_VEL
LIN {X 0,Y 165.138,Z 422.44,A -85,B 0,C 180,E1 -23906.501,E2 -23906.501} C_VEL
LIN {X 0,Y 156.952,Z 408.221,A -85,B 0,C 180,E1 -23910.03,E2 -23910.03} C_VEL
LIN {X 0,Y 152.696,Z 401.107,A -85,B 0,C 180,E1 -23912.038,E2 -23912.038} C_VEL
LIN {X 0,Y 150.731,Z 398.245,A -85,B 0,C 180,E1 -23912.988,E2 -23912.988} C_VEL
LIN {X 0,Y 150.232,Z 396.385,A -85,B 0,C 180,E1 -23913.398,E2 -23913.398} C_VEL
LIN {X 0,Y 150.27,Z 396.383,A -85,B 0,C 180,E1 -23919.277,E2 -23919.277} C_VEL
LIN {X 0,Y 150.303,Z 396.385,A -85,B 0,C 180,E1 -23923.707,E2 -23923.707} C_VEL
LIN {X 0,Y 150.593,Z 396.325,A -85,B 0,C 180,E1 -23929.242,E2 -23929.242} C_VEL
LIN {X 0,Y 150.667,Z 396.331,A -85,B 0,C 180,E1 -23931.956,E2 -23931.956} C_VEL
LIN {X 0,Y 151.184,Z 396.28,A -85,B 0,C 180,E1 -23940.001,E2 -23940.001} C_VEL
LIN {X 0,Y 150.669,Z 396.339,A -85,B 0,C 180,E1 -23948.045,E2 -23948.045} C_VEL
LIN {X 0,Y 150.561,Z 396.348,A -85,B 0,C 180,E1 -23951.429,E2 -23951.429} C_VEL
LIN {X 0,Y 150.303,Z 396.379,A -85,B 0,C 180,E1 -23956.294,E2 -23956.294} C_VEL
LIN {X 0,Y 150.271,Z 396.391,A -85,B 0,C 180,E1 -23960.724,E2 -23960.724} C_VEL
LIN {X 0,Y 150.175,Z 396.395,A -85,B 0,C 180,E1 -23967.24,E2 -23967.24} C_VEL
LIN {X 0,Y 150.199,Z 396.392,A -85,B 0,C 180,E1 -23972.631,E2 -23972.631} C_VEL
LIN {X 0,Y 150.161,Z 396.403,A -85,B 0,C 180,E1 -23977.478,E2 -23977.478} C_VEL
LIN {X 0,Y 150.125,Z 396.397,A -85,B 0,C 180,E1 -23981.5,E2 -23981.5} C_VEL
LIN {X 0,Y 150.12,Z 396.407,A -85,B 0,C 180,E1 -23985.399,E2 -23985.399} C_VEL
LIN {X 0,Y 150.13,Z 396.402,A -85,B 0,C 180,E1 -23989.058,E2 -23989.058} C_VEL
LIN {X 0,Y 150.17,Z 396.4,A -85,B 0,C 180,E1 -23992.714,E2 -23992.714} C_VEL
LIN {X 0,Y 150.201,Z 396.392,A -85,B 0,C 180,E1 -23997.378,E2 -23997.378} C_VEL
LIN {X 0,Y 150.235,Z 396.396,A -85,B 0,C 180,E1 -24002.727,E2 -24002.727} C_VEL
LIN {X 0,Y 150.284,Z 396.392,A -85,B 0,C 180,E1 -24009.278,E2 -24009.278} C_VEL
LIN {X 0,Y 150.324,Z 396.353,A -85,B 0,C 180,E1 -24013.714,E2 -24013.714} C_VEL
LIN {X 0,Y 150.608,Z 396.347,A -85,B 0,C 180,E1 -24019.246,E2 -24019.246} C_VEL
LIN {X 0,Y 150.682,Z 396.335,A -85,B 0,C 180,E1 -24021.961,E2 -24021.961} C_VEL
LIN {X 0,Y 151.2,Z 396.277,A -85,B 0,C 180,E1 -24030.004,E2 -24030.004} C_VEL
LIN {X 0,Y 150.662,Z 396.333,A -85,B 0,C 180,E1 -24038.639,E2 -24038.639} C_VEL
LIN {X 0,Y 151.614,Z 399.128,A -85,B 0,C 180,E1 -24039.257,E2 -24039.257} C_VEL
LIN {X 0,Y 153.192,Z 401.28,A -85,B 0,C 180,E1 -24039.994,E2 -24039.994} C_VEL
LIN {X 0,Y 163.534,Z 419.434,A -85,B 0,C 180,E1 -24044.645,E2 -24044.645} C_VEL
LIN {X 0,Y 172.802,Z 437.165,A -85,B 0,C 180,E1 -24048.404,E2 -24048.404} C_VEL
LIN {X 0,Y 182.693,Z 457.87,A -85,B 0,C 180,E1 -24052.029,E2 -24052.029} C_VEL
LIN {X 0,Y 185.529,Z 464.326,A -85,B 0,C 180,E1 -24053.023,E2 -24053.023} C_VEL
LIN {X 0,Y 176.83,Z 547.578,A -85,B 0,C 180,E1 -24057.371,E2 -24057.371} C_VEL
LIN {X 0,Y 174.509,Z 563.727,A -85,B 0,C 180,E1 -24058.655,E2 -24058.655} C_VEL
LIN {X 0,Y 171.618,Z 579.943,A -85,B 0,C 180,E1 -24060.432,E2 -24060.432} C_VEL
LIN {X 0,Y 168.421,Z 594.718,A -85,B 0,C 180,E1 -24062.537,E2 -24062.537} C_VEL
LIN {X 0,Y 164.713,Z 609.855,A -85,B 0,C 180,E1 -24065.31,E2 -24065.31} C_VEL
LIN {X 0,Y 161.209,Z 622.853,A -85,B 0,C 180,E1 -24068.304,E2 -24068.304} C_VEL
LIN {X 0,Y 157.634,Z 635.683,A -85,B 0,C 180,E1 -24071.976,E2 -24071.976} C_VEL
LIN {X 0,Y 154.445,Z 647.136,A -85,B 0,C 180,E1 -24076.055,E2 -24076.055} C_VEL
LIN {X 0,Y 151.799,Z 657.094,A -85,B 0,C 180,E1 -24080.428,E2 -24080.428} C_VEL
LIN {X 0,Y 149.852,Z 665.47,A -85,B 0,C 180,E1 -24084.933,E2 -24084.933} C_VEL
LIN {X 0,Y 148.465,Z 673.387,A -85,B 0,C 180,E1 -24090.194,E2 -24090.194} C_VEL
LIN {X 0,Y 147.651,Z 678.798,A -85,B 0,C 180,E1 -24094.747,E2 -24094.747} C_VEL
LIN {X 0,Y 147.18,Z 684.148,A -85,B 0,C 180,E1 -24100.472,E2 -24100.472} C_VEL
LIN {X 0,Y 147.297,Z 686.298,A -85,B 0,C 180,E1 -24103.364,E2 -24103.364} C_VEL
LIN {X 0,Y 147.942,Z 689.514,A -85,B 0,C 180,E1 -24109.045,E2 -24109.045} C_VEL
LIN {X 0,Y 149.722,Z 691.521,A -85,B 0,C 180,E1 -24114.612,E2 -24114.612} C_VEL
LIN {X 0,Y 152.547,Z 692.404,A -85,B 0,C 180,E1 -24119.999,E2 -24119.999} C_VEL
LIN {X 0,Y 156.592,Z 692.177,A -85,B 0,C 180,E1 -24125.149,E2 -24125.149} C_VEL
LIN {X 0,Y 161.878,Z 690.936,A -85,B 0,C 180,E1 -24130,E2 -24130} C_VEL
LIN {X 0,Y 168.285,Z 688.688,A -85,B 0,C 180,E1 -24134.511,E2 -24134.511} C_VEL
LIN {X 0,Y 177.793,Z 684.313,A -85,B 0,C 180,E1 -24139.633,E2 -24139.633} C_VEL
LIN {X 0,Y 186.582,Z 679.523,A -85,B 0,C 180,E1 -24143.297,E2 -24143.297} C_VEL
LIN {X 0,Y 196.835,Z 673.098,A -85,B 0,C 180,E1 -24146.789,E2 -24146.789} C_VEL
LIN {X 0,Y 207.993,Z 665.11,A -85,B 0,C 180,E1 -24149.893,E2 -24149.893} C_VEL
LIN {X 0,Y 219.256,Z 655.891,A -85,B 0,C 180,E1 -24152.473,E2 -24152.473} C_VEL
LIN {X 0,Y 228.971,Z 646.928,A -85,B 0,C 180,E1 -24154.379,E2 -24154.379} C_VEL
LIN {X 0,Y 230.891,Z 645.019,A -85,B 0,C 180,E1 -24154.727,E2 -24154.727} C_VEL
LIN {X 0,Y 231.478,Z 644.414,A -85,B 0,C 180,E1 -24154.936,E2 -24154.936} C_VEL
LIN {X 0,Y 221.328,Z 654.402,A -85,B 0,C 180,E1 -24156.696,E2 -24156.696} C_VEL
LIN {X 0,Y 208.977,Z 665.181,A -85,B 0,C 180,E1 -24159.327,E2 -24159.327} C_VEL
LIN {X 0,Y 198.556,Z 673.248,A -85,B 0,C 180,E1 -24162.014,E2 -24162.014} C_VEL
LIN {X 0,Y 194.458,Z 676.088,A -85,B 0,C 180,E1 -24162.954,E2 -24162.954} C_VEL
LIN {X 0,Y 186.668,Z 680.646,A -85,B 0,C 180,E1 -24164.202,E2 -24164.202} C_VEL
LIN {X 0,Y 178.871,Z 684.694,A -85,B 0,C 180,E1 -24165.615,E2 -24165.615} C_VEL
LIN {X 0,Y 174.839,Z 686.73,A -85,B 0,C 180,E1 -24166.827,E2 -24166.827} C_VEL
LIN {X 0,Y 166.434,Z 691.029,A -85,B 0,C 180,E1 -24170.694,E2 -24170.694} C_VEL
LIN {X 0,Y 159.204,Z 694.259,A -85,B 0,C 180,E1 -24174.975,E2 -24174.975} C_VEL
LIN {X 0,Y 152.942,Z 696.564,A -85,B 0,C 180,E1 -24179.633,E2 -24179.633} C_VEL
LIN {X 0,Y 147.664,Z 697.971,A -85,B 0,C 180,E1 -24184.727,E2 -24184.727} C_VEL
LIN {X 0,Y 144.188,Z 698.331,A -85,B 0,C 180,E1 -24190.046,E2 -24190.046} C_VEL
LIN {X 0,Y 141.874,Z 697.775,A -85,B 0,C 180,E1 -24195.655,E2 -24195.655} C_VEL
LIN {X 0,Y 140.837,Z 696.197,A -85,B 0,C 180,E1 -24201.386,E2 -24201.386} C_VEL
LIN {X 0,Y 140.945,Z 693.494,A -85,B 0,C 180,E1 -24207.138,E2 -24207.138} C_VEL
LIN {X 0,Y 141.065,Z 690.623,A -85,B 0,C 180,E1 -24211.423,E2 -24211.423} C_VEL
LIN {X 0,Y 141.074,Z 686.809,A -85,B 0,C 180,E1 -24215.714,E2 -24215.714} C_VEL
LIN {X 0,Y 141.316,Z 682.136,A -85,B 0,C 180,E1 -24220.02,E2 -24220.02} C_VEL
LIN {X 0,Y 142.402,Z 674.354,A -85,B 0,C 180,E1 -24225.746,E2 -24225.746} C_VEL
LIN {X 0,Y 144.226,Z 665.863,A -85,B 0,C 180,E1 -24230.684,E2 -24230.684} C_VEL
LIN {X 0,Y 146.988,Z 655.617,A -85,B 0,C 180,E1 -24235.483,E2 -24235.483} C_VEL
LIN {X 0,Y 149.942,Z 645.079,A -85,B 0,C 180,E1 -24239.477,E2 -24239.477} C_VEL
LIN {X 0,Y 153.596,Z 632.567,A -85,B 0,C 180,E1 -24243.299,E2 -24243.299} C_VEL
LIN {X 0,Y 157.187,Z 619.868,A -85,B 0,C 180,E1 -24246.41,E2 -24246.41} C_VEL
LIN {X 0,Y 161.004,Z 605.178,A -85,B 0,C 180,E1 -24249.262,E2 -24249.262} C_VEL
LIN {X 0,Y 164.687,Z 589.519,A -85,B 0,C 180,E1 -24251.61,E2 -24251.61} C_VEL
LIN {X 0,Y 167.652,Z 574.393,A -85,B 0,C 180,E1 -24253.344,E2 -24253.344} C_VEL
LIN {X 0,Y 170.314,Z 557.801,A -85,B 0,C 180,E1 -24254.729,E2 -24254.729} C_VEL
LIN {X 0,Y 175.273,Z 511.209,A -85,B 0,C 180,E1 -24257.347,E2 -24257.347} C_VEL
LIN {X 0,Y 179.228,Z 473.675,A -85,B 0,C 180,E1 -24259.326,E2 -24259.326} C_VEL
LIN {X 0,Y 172.484,Z 455.829,A -85,B 0,C 180,E1 -24262.048,E2 -24262.048} C_VEL
LIN {X 0,Y 164.249,Z 435.52,A -85,B 0,C 180,E1 -24265.626,E2 -24265.626} C_VEL
LIN {X 0,Y 159.955,Z 426.407,A -85,B 0,C 180,E1 -24267.542,E2 -24267.542} C_VEL
LIN {X 0,Y 152.407,Z 413.122,A -85,B 0,C 180,E1 -24270.959,E2 -24270.959} C_VEL
LIN {X 0,Y 147.477,Z 405.104,A -85,B 0,C 180,E1 -24273.4,E2 -24273.4} C_VEL
LIN {X 0,Y 145.205,Z 401.446,A -85,B 0,C 180,E1 -24274.562,E2 -24274.562} C_VEL
LIN {X 0,Y 143.569,Z 399.016,A -85,B 0,C 180,E1 -24275.413,E2 -24275.413} C_VEL
LIN {X 0,Y 143.101,Z 397.276,A -85,B 0,C 180,E1 -24275.81,E2 -24275.81} C_VEL
LIN {X 0,Y 143.234,Z 397.253,A -85,B 0,C 180,E1 -24279.913,E2 -24279.913} C_VEL
LIN {X 0,Y 143.294,Z 397.261,A -85,B 0,C 180,E1 -24285.805,E2 -24285.805} C_VEL
LIN {X 0,Y 143.519,Z 397.207,A -85,B 0,C 180,E1 -24288.705,E2 -24288.705} C_VEL
LIN {X 0,Y 143.593,Z 397.207,A -85,B 0,C 180,E1 -24291.557,E2 -24291.557} C_VEL
LIN {X 0,Y 144.142,Z 397.157,A -85,B 0,C 180,E1 -24300.001,E2 -24300.001} C_VEL
LIN {X 0,Y 143.595,Z 397.219,A -85,B 0,C 180,E1 -24308.444,E2 -24308.444} C_VEL
LIN {X 0,Y 143.486,Z 397.23,A -85,B 0,C 180,E1 -24311.616,E2 -24311.616} C_VEL
LIN {X 0,Y 143.242,Z 397.255,A -85,B 0,C 180,E1 -24317.121,E2 -24317.121} C_VEL
LIN {X 0,Y 143.208,Z 397.271,A -85,B 0,C 180,E1 -24321.196,E2 -24321.196} C_VEL
LIN {X 0,Y 143.132,Z 397.275,A -85,B 0,C 180,E1 -24327.903,E2 -24327.903} C_VEL
LIN {X 0,Y 143.129,Z 397.267,A -85,B 0,C 180,E1 -24333.419,E2 -24333.419} C_VEL
LIN {X 0,Y 143.044,Z 397.288,A -85,B 0,C 180,E1 -24339.697,E2 -24339.697} C_VEL
LIN {X 0,Y 143.026,Z 397.281,A -85,B 0,C 180,E1 -24343.468,E2 -24343.468} C_VEL
LIN {X 0,Y 143.031,Z 397.293,A -85,B 0,C 180,E1 -24347.482,E2 -24347.482} C_VEL
LIN {X 0,Y 143.065,Z 397.277,A -85,B 0,C 180,E1 -24351.814,E2 -24351.814} C_VEL
LIN {X 0,Y 143.168,Z 397.267,A -85,B 0,C 180,E1 -24357.323,E2 -24357.323} C_VEL
LIN {X 0,Y 143.179,Z 397.276,A -85,B 0,C 180,E1 -24362.074,E2 -24362.074} C_VEL
LIN {X 0,Y 143.225,Z 397.27,A -85,B 0,C 180,E1 -24368.803,E2 -24368.803} C_VEL
LIN {X 0,Y 143.261,Z 397.239,A -85,B 0,C 180,E1 -24372.886,E2 -24372.886} C_VEL
LIN {X 0,Y 143.535,Z 397.225,A -85,B 0,C 180,E1 -24378.71,E2 -24378.71} C_VEL
LIN {X 0,Y 143.608,Z 397.218,A -85,B 0,C 180,E1 -24381.562,E2 -24381.562} C_VEL
LIN {X 0,Y 144.159,Z 397.154,A -85,B 0,C 180,E1 -24390.004,E2 -24390.004} C_VEL
LIN {X 0,Y 143.59,Z 397.229,A -85,B 0,C 180,E1 -24396.239,E2 -24396.239} C_VEL
LIN {X 0,Y 144.653,Z 400.163,A -85,B 0,C 180,E1 -24396.981,E2 -24396.981} C_VEL
LIN {X 0,Y 146.27,Z 402.243,A -85,B 0,C 180,E1 -24397.771,E2 -24397.771} C_VEL
LIN {X 0,Y 150.964,Z 410.344,A -85,B 0,C 180,E1 -24400.155,E2 -24400.155} C_VEL
LIN {X 0,Y 158.594,Z 423.808,A -85,B 0,C 180,E1 -24403.709,E2 -24403.709} C_VEL
LIN {X 0,Y 166.573,Z 439.133,A -85,B 0,C 180,E1 -24407.094,E2 -24407.094} C_VEL
LIN {X 0,Y 176.794,Z 460.559,A -85,B 0,C 180,E1 -24411.027,E2 -24411.027} C_VEL
LIN {X 0,Y 179.284,Z 466.471,A -85,B 0,C 180,E1 -24411.969,E2 -24411.969} C_VEL
LIN {X 0,Y 170.521,Z 547.124,A -85,B 0,C 180,E1 -24416.308,E2 -24416.308} C_VEL
LIN {X 0,Y 168.04,Z 563.853,A -85,B 0,C 180,E1 -24417.683,E2 -24417.683} C_VEL
LIN {X 0,Y 165.05,Z 579.966,A -85,B 0,C 180,E1 -24419.51,E2 -24419.51} C_VEL
LIN {X 0,Y 161.676,Z 595.019,A -85,B 0,C 180,E1 -24421.739,E2 -24421.739} C_VEL
LIN {X 0,Y 157.896,Z 609.954,A -85,B 0,C 180,E1 -24424.57,E2 -24424.57} C_VEL
LIN {X 0,Y 154.305,Z 622.987,A -85,B 0,C 180,E1 -24427.686,E2 -24427.686} C_VEL
LIN {X 0,Y 151.004,Z 634.508,A -85,B 0,C 180,E1 -24431.086,E2 -24431.086} C_VEL
LIN {X 0,Y 147.677,Z 645.997,A -85,B 0,C 180,E1 -24435.247,E2 -24435.247} C_VEL
LIN {X 0,Y 144.815,Z 656.534,A -85,B 0,C 180,E1 -24439.98,E2 -24439.98} C_VEL
LIN {X 0,Y 142.815,Z 664.925,A -85,B 0,C 180,E1 -24444.673,E2 -24444.673} C_VEL
LIN {X 0,Y 141.691,Z 670.943,A -85,B 0,C 180,E1 -24448.705,E2 -24448.705} C_VEL
LIN {X 0,Y 140.7,Z 677.519,A -85,B 0,C 180,E1 -24454.049,E2 -24454.049} C_VEL
LIN {X 0,Y 140.153,Z 682.751,A -85,B 0,C 180,E1 -24459.45,E2 -24459.45} C_VEL
LIN {X 0,Y 140.164,Z 685.131,A -85,B 0,C 180,E1 -24462.491,E2 -24462.491} C_VEL
LIN {X 0,Y 140.707,Z 688.756,A -85,B 0,C 180,E1 -24468.474,E2 -24468.474} C_VEL
LIN {X 0,Y 142.441,Z 691.169,A -85,B 0,C 180,E1 -24474.336,E2 -24474.336} C_VEL
LIN {X 0,Y 145.25,Z 692.454,A -85,B 0,C 180,E1 -24479.999,E2 -24479.999} C_VEL
LIN {X 0,Y 149.338,Z 692.698,A -85,B 0,C 180,E1 -24485.4,E2 -24485.4} C_VEL
LIN {X 0,Y 154.749,Z 691.855,A -85,B 0,C 180,E1 -24490.466,E2 -24490.466} C_VEL
LIN {X 0,Y 161.288,Z 690.022,A -85,B 0,C 180,E1 -24495.155,E2 -24495.155} C_VEL
LIN {X 0,Y 168.967,Z 687.191,A -85,B 0,C 180,E1 -24499.435,E2 -24499.435} C_VEL
LIN {X 0,Y 177.692,Z 683.197,A -85,B 0,C 180,E1 -24503.298,E2 -24503.298} C_VEL
LIN {X 0,Y 187.371,Z 678.032,A -85,B 0,C 180,E1 -24506.75,E2 -24506.75} C_VEL
LIN {X 0,Y 197.794,Z 671.69,A -85,B 0,C 180,E1 -24509.831,E2 -24509.831} C_VEL
LIN {X 0,Y 210.47,Z 662.782,A -85,B 0,C 180,E1 -24512.862,E2 -24512.862} C_VEL
LIN {X 0,Y 218.841,Z 656.174,A -85,B 0,C 180,E1 -24514.542,E2 -24514.542} C_VEL
LIN {X 0,Y 217.634,Z 657.226,A -85,B 0,C 180,E1 -24515.255,E2 -24515.255} C_VEL
LIN {X 0,Y 206.129,Z 666.543,A -85,B 0,C 180,E1 -24517.556,E2 -24517.556} C_VEL
LIN {X 0,Y 194.102,Z 675.155,A -85,B 0,C 180,E1 -24520.5,E2 -24520.5} C_VEL
LIN {X 0,Y 184.054,Z 681.511,A -85,B 0,C 180,E1 -24523.485,E2 -24523.485} C_VEL
LIN {X 0,Y 174.839,Z 686.73,A -85,B 0,C 180,E1 -24526.827,E2 -24526.827} C_VEL
LIN {X 0,Y 170.864,Z 688.645,A -85,B 0,C 180,E1 -24528.139,E2 -24528.139} C_VEL
LIN {X 0,Y 163.294,Z 691.549,A -85,B 0,C 180,E1 -24530.1,E2 -24530.1} C_VEL
LIN {X 0,Y 157.352,Z 693.481,A -85,B 0,C 180,E1 -24531.824,E2 -24531.824} C_VEL
LIN {X 0,Y 153.57,Z 694.674,A -85,B 0,C 180,E1 -24533.423,E2 -24533.423} C_VEL
LIN {X 0,Y 152.542,Z 694.989,A -85,B 0,C 180,E1 -24534.034,E2 -24534.034} C_VEL
LIN {X 0,Y 146.832,Z 696.73,A -85,B 0,C 180,E1 -24538.226,E2 -24538.226} C_VEL
LIN {X 0,Y 140.962,Z 697.866,A -85,B 0,C 180,E1 -24543.821,E2 -24543.821} C_VEL
LIN {X 0,Y 137.475,Z 698.032,A -85,B 0,C 180,E1 -24549.027,E2 -24549.027} C_VEL
LIN {X 0,Y 134.989,Z 697.207,A -85,B 0,C 180,E1 -24554.907,E2 -24554.907} C_VEL
LIN {X 0,Y 133.841,Z 695.418,A -85,B 0,C 180,E1 -24560.932,E2 -24560.932} C_VEL
LIN {X 0,Y 133.906,Z 692.554,A -85,B 0,C 180,E1 -24566.987,E2 -24566.987} C_VEL
LIN {X 0,Y 134.048,Z 689.484,A -85,B 0,C 180,E1 -24571.498,E2 -24571.498} C_VEL
LIN {X 0,Y 134.036,Z 685.505,A -85,B 0,C 180,E1 -24576.015,E2 -24576.015} C_VEL
LIN {X 0,Y 134.338,Z 680.582,A -85,B 0,C 180,E1 -24580.546,E2 -24580.546} C_VEL
LIN {X 0,Y 135.351,Z 673.589,A -85,B 0,C 180,E1 -24585.814,E2 -24585.814} C_VEL
LIN {X 0,Y 137.242,Z 665.068,A -85,B 0,C 180,E1 -24591.001,E2 -24591.001} C_VEL
LIN {X 0,Y 140.094,Z 654.743,A -85,B 0,C 180,E1 -24596.039,E2 -24596.039} C_VEL
LIN {X 0,Y 143.138,Z 644.138,A -85,B 0,C 180,E1 -24600.211,E2 -24600.211} C_VEL
LIN {X 0,Y 146.974,Z 631.492,A -85,B 0,C 180,E1 -24604.179,E2 -24604.179} C_VEL
LIN {X 0,Y 150.601,Z 618.917,A -85,B 0,C 180,E1 -24607.343,E2 -24607.343} C_VEL
LIN {X 0,Y 154.223,Z 605.402,A -85,B 0,C 180,E1 -24610.061,E2 -24610.061} C_VEL
LIN {X 0,Y 158.002,Z 589.842,A -85,B 0,C 180,E1 -24612.491,E2 -24612.491} C_VEL
LIN {X 0,Y 161.3,Z 573.591,A -85,B 0,C 180,E1 -24614.41,E2 -24614.41} C_VEL
LIN {X 0,Y 163.931,Z 557.525,A -85,B 0,C 180,E1 -24615.782,E2 -24615.782} C_VEL
LIN {X 0,Y 169.929,Z 502.98,A -85,B 0,C 180,E1 -24618.949,E2 -24618.949} C_VEL
LIN {X 0,Y 173.014,Z 475.397,A -85,B 0,C 180,E1 -24620.444,E2 -24620.444} C_VEL
LIN {X 0,Y 165.347,Z 455.04,A -85,B 0,C 180,E1 -24623.714,E2 -24623.714} C_VEL
LIN {X 0,Y 157.829,Z 436.727,A -85,B 0,C 180,E1 -24627.198,E2 -24627.198} C_VEL
LIN {X 0,Y 154.697,Z 430.169,A -85,B 0,C 180,E1 -24628.654,E2 -24628.654} C_VEL
LIN {X 0,Y 147.672,Z 417.613,A -85,B 0,C 180,E1 -24632.065,E2 -24632.065} C_VEL
LIN {X 0,Y 141.008,Z 406.687,A -85,B 0,C 180,E1 -24635.525,E2 -24635.525} C_VEL
LIN {X 0,Y 138.945,Z 403.395,A -85,B 0,C 180,E1 -24636.695,E2 -24636.695} C_VEL
LIN {X 0,Y 136.68,Z 400.238,A -85,B 0,C 180,E1 -24637.992,E2 -24637.992} C_VEL
LIN {X 0,Y 136.145,Z 398.148,A -85,B 0,C 180,E1 -24638.562,E2 -24638.562} C_VEL
LIN {X 0,Y 136.212,Z 398.145,A -85,B 0,C 180,E1 -24645.051,E2 -24645.051} C_VEL
LIN {X 0,Y 136.413,Z 398.094,A -85,B 0,C 180,E1 -24648.178,E2 -24648.178} C_VEL
LIN {X 0,Y 136.522,Z 398.082,A -85,B 0,C 180,E1 -24651.117,E2 -24651.117} C_VEL
LIN {X 0,Y 137.099,Z 398.034,A -85,B 0,C 180,E1 -24660.001,E2 -24660.001} C_VEL
LIN {X 0,Y 136.524,Z 398.097,A -85,B 0,C 180,E1 -24668.885,E2 -24668.885} C_VEL
LIN {X 0,Y 136.402,Z 398.113,A -85,B 0,C 180,E1 -24671.895,E2 -24671.895} C_VEL
LIN {X 0,Y 136.154,Z 398.137,A -85,B 0,C 180,E1 -24678.043,E2 -24678.043} C_VEL
LIN {X 0,Y 136.133,Z 398.153,A -85,B 0,C 180,E1 -24681.692,E2 -24681.692} C_VEL
LIN {X 0,Y 136.052,Z 398.161,A -85,B 0,C 180,E1 -24688.589,E2 -24688.589} C_VEL
LIN {X 0,Y 136.031,Z 398.15,A -85,B 0,C 180,E1 -24694.634,E2 -24694.634} C_VEL
LIN {X 0,Y 136.016,Z 398.166,A -85,B 0,C 180,E1 -24699.198,E2 -24699.198} C_VEL
LIN {X 0,Y 135.971,Z 398.16,A -85,B 0,C 180,E1 -24703.652,E2 -24703.652} C_VEL
LIN {X 0,Y 135.975,Z 398.17,A -85,B 0,C 180,E1 -24707.792,E2 -24707.792} C_VEL
LIN {X 0,Y 136.014,Z 398.154,A -85,B 0,C 180,E1 -24711.686,E2 -24711.686} C_VEL
LIN {X 0,Y 136.047,Z 398.162,A -85,B 0,C 180,E1 -24715.747,E2 -24715.747} C_VEL
LIN {X 0,Y 136.135,Z 398.153,A -85,B 0,C 180,E1 -24722.319,E2 -24722.319} C_VEL
LIN {X 0,Y 136.189,Z 398.147,A -85,B 0,C 180,E1 -24728.829,E2 -24728.829} C_VEL
LIN {X 0,Y 136.232,Z 398.102,A -85,B 0,C 180,E1 -24735.057,E2 -24735.057} C_VEL
LIN {X 0,Y 136.426,Z 398.105,A -85,B 0,C 180,E1 -24738.182,E2 -24738.182} C_VEL
LIN {X 0,Y 136.537,Z 398.102,A -85,B 0,C 180,E1 -24741.121,E2 -24741.121} C_VEL
LIN {X 0,Y 137.115,Z 398.031,A -85,B 0,C 180,E1 -24750.004,E2 -24750.004} C_VEL
LIN {X 0,Y 136.641,Z 398.076,A -85,B 0,C 180,E1 -24753.598,E2 -24753.598} C_VEL
LIN {X 0,Y 137.688,Z 401.07,A -85,B 0,C 180,E1 -24754.395,E2 -24754.395} C_VEL
LIN {X 0,Y 139.396,Z 403.257,A -85,B 0,C 180,E1 -24755.338,E2 -24755.338} C_VEL
LIN {X 0,Y 141.306,Z 406.443,A -85,B 0,C 180,E1 -24756.429,E2 -24756.429} C_VEL
LIN {X 0,Y 145.954,Z 414.209,A -85,B 0,C 180,E1 -24758.897,E2 -24758.897} C_VEL
LIN {X 0,Y 153.814,Z 428.46,A -85,B 0,C 180,E1 -24762.78,E2 -24762.78} C_VEL
LIN {X 0,Y 161.474,Z 443.314,A -85,B 0,C 180,E1 -24766.162,E2 -24766.162} C_VEL
LIN {X 0,Y 171.273,Z 464.16,A -85,B 0,C 180,E1 -24770.166,E2 -24770.166} C_VEL
LIN {X 0,Y 172.994,Z 468.659,A -85,B 0,C 180,E1 -24770.868,E2 -24770.868} C_VEL
LIN {X 0,Y 164.061,Z 547.619,A -85,B 0,C 180,E1 -24775.268,E2 -24775.268} C_VEL
LIN {X 0,Y 161.645,Z 563.57,A -85,B 0,C 180,E1 -24776.616,E2 -24776.616} C_VEL
LIN {X 0,Y 158.556,Z 579.807,A -85,B 0,C 180,E1 -24778.503,E2 -24778.503} C_VEL
LIN {X 0,Y 155.252,Z 594.158,A -85,B 0,C 180,E1 -24780.671,E2 -24780.671} C_VEL
LIN {X 0,Y 151.572,Z 608.457,A -85,B 0,C 180,E1 -24783.423,E2 -24783.423} C_VEL
LIN {X 0,Y 147.781,Z 621.836,A -85,B 0,C 180,E1 -24786.662,E2 -24786.662} C_VEL
LIN {X 0,Y 144.155,Z 634.093,A -85,B 0,C 180,E1 -24790.378,E2 -24790.378} C_VEL
LIN {X 0,Y 140.656,Z 645.881,A -85,B 0,C 180,E1 -24794.84,E2 -24794.84} C_VEL
LIN {X 0,Y 137.888,Z 655.745,A -85,B 0,C 180,E1 -24799.467,E2 -24799.467} C_VEL
LIN {X 0,Y 135.781,Z 664.301,A -85,B 0,C 180,E1 -24804.387,E2 -24804.387} C_VEL
LIN {X 0,Y 134.479,Z 671.42,A -85,B 0,C 180,E1 -24809.365,E2 -24809.365} C_VEL
LIN {X 0,Y 133.768,Z 676.106,A -85,B 0,C 180,E1 -24813.281,E2 -24813.281} C_VEL
LIN {X 0,Y 133.159,Z 681.068,A -85,B 0,C 180,E1 -24818.317,E2 -24818.317} C_VEL
LIN {X 0,Y 133.084,Z 683.987,A -85,B 0,C 180,E1 -24821.92,E2 -24821.92} C_VEL
LIN {X 0,Y 133.513,Z 687.846,A -85,B 0,C 180,E1 -24827.844,E2 -24827.844} C_VEL
LIN {X 0,Y 135.173,Z 690.68,A -85,B 0,C 180,E1 -24834.03,E2 -24834.03} C_VEL
LIN {X 0,Y 137.934,Z 692.348,A -85,B 0,C 180,E1 -24839.999,E2 -24839.999} C_VEL
LIN {X 0,Y 142.101,Z 692.997,A -85,B 0,C 180,E1 -24845.676,E2 -24845.676} C_VEL
LIN {X 0,Y 147.609,Z 692.637,A -85,B 0,C 180,E1 -24850.978,E2 -24850.978} C_VEL
LIN {X 0,Y 154.331,Z 691.222,A -85,B 0,C 180,E1 -24855.856,E2 -24855.856} C_VEL
LIN {X 0,Y 162.182,Z 688.819,A -85,B 0,C 180,E1 -24860.283,E2 -24860.283} C_VEL
LIN {X 0,Y 171.127,Z 685.409,A -85,B 0,C 180,E1 -24864.247,E2 -24864.247} C_VEL
LIN {X 0,Y 181.015,Z 680.804,A -85,B 0,C 180,E1 -24867.768,E2 -24867.768} C_VEL
LIN {X 0,Y 191.682,Z 675.026,A -85,B 0,C 180,E1 -24870.884,E2 -24870.884} C_VEL
LIN {X 0,Y 203.16,Z 667.924,A -85,B 0,C 180,E1 -24873.606,E2 -24873.606} C_VEL
LIN {X 0,Y 207.219,Z 665.175,A -85,B 0,C 180,E1 -24874.466,E2 -24874.466} C_VEL
LIN {X 0,Y 206.362,Z 665.85,A -85,B 0,C 180,E1 -24875.174,E2 -24875.174} C_VEL
LIN {X 0,Y 195.12,Z 673.573,A -85,B 0,C 180,E1 -24877.584,E2 -24877.584} C_VEL
LIN {X 0,Y 183.279,Z 680.756,A -85,B 0,C 180,E1 -24880.683,E2 -24880.683} C_VEL
LIN {X 0,Y 172.051,Z 686.694,A -85,B 0,C 180,E1 -24884.365,E2 -24884.365} C_VEL
LIN {X 0,Y 165.238,Z 689.93,A -85,B 0,C 180,E1 -24887.111,E2 -24887.111} C_VEL
LIN {X 0,Y 157.09,Z 693.322,A -85,B 0,C 180,E1 -24891.215,E2 -24891.215} C_VEL
LIN {X 0,Y 152.542,Z 694.989,A -85,B 0,C 180,E1 -24894.034,E2 -24894.034} C_VEL
LIN {X 0,Y 149.156,Z 695.946,A -85,B 0,C 180,E1 -24895.845,E2 -24895.845} C_VEL
LIN {X 0,Y 142.322,Z 697.078,A -85,B 0,C 180,E1 -24898.645,E2 -24898.645} C_VEL
LIN {X 0,Y 135.943,Z 697.663,A -85,B 0,C 180,E1 -24901.752,E2 -24901.752} C_VEL
LIN {X 0,Y 133.374,Z 697.741,A -85,B 0,C 180,E1 -24904.006,E2 -24904.006} C_VEL
LIN {X 0,Y 129.247,Z 697.224,A -85,B 0,C 180,E1 -24910.953,E2 -24910.953} C_VEL
LIN {X 0,Y 127.306,Z 695.724,A -85,B 0,C 180,E1 -24917.238,E2 -24917.238} C_VEL
LIN {X 0,Y 126.734,Z 693.18,A -85,B 0,C 180,E1 -24923.628,E2 -24923.628} C_VEL
LIN {X 0,Y 126.927,Z 690.829,A -85,B 0,C 180,E1 -24927.888,E2 -24927.888} C_VEL
LIN {X 0,Y 127.05,Z 688.256,A -85,B 0,C 180,E1 -24931.58,E2 -24931.58} C_VEL
LIN {X 0,Y 127.03,Z 684.115,A -85,B 0,C 180,E1 -24936.348,E2 -24936.348} C_VEL
LIN {X 0,Y 127.384,Z 678.983,A -85,B 0,C 180,E1 -24941.129,E2 -24941.129} C_VEL
LIN {X 0,Y 128.507,Z 671.661,A -85,B 0,C 180,E1 -24946.681,E2 -24946.681} C_VEL
LIN {X 0,Y 130.638,Z 662.796,A -85,B 0,C 180,E1 -24952.117,E2 -24952.117} C_VEL
LIN {X 0,Y 133.646,Z 652.233,A -85,B 0,C 180,E1 -24957.305,E2 -24957.305} C_VEL
LIN {X 0,Y 136.965,Z 641.003,A -85,B 0,C 180,E1 -24961.727,E2 -24961.727} C_VEL
LIN {X 0,Y 140.736,Z 629.099,A -85,B 0,C 180,E1 -24965.482,E2 -24965.482} C_VEL
LIN {X 0,Y 144.479,Z 616.361,A -85,B 0,C 180,E1 -24968.714,E2 -24968.714} C_VEL
LIN {X 0,Y 148.354,Z 602.255,A -85,B 0,C 180,E1 -24971.54,E2 -24971.54} C_VEL
LIN {X 0,Y 152.079,Z 587.094,A -85,B 0,C 180,E1 -24973.877,E2 -24973.877} C_VEL
LIN {X 0,Y 155.284,Z 571.539,A -85,B 0,C 180,E1 -24975.691,E2 -24975.691} C_VEL
LIN {X 0,Y 157.838,Z 555.634,A -85,B 0,C 180,E1 -24977.04,E2 -24977.04} C_VEL
LIN {X 0,Y 166.757,Z 477.052,A -85,B 0,C 180,E1 -24981.608,E2 -24981.608} C_VEL
LIN {X 0,Y 159.764,Z 458.166,A -85,B 0,C 180,E1 -24984.832,E2 -24984.832} C_VEL
LIN {X 0,Y 151.886,Z 438.716,A -85,B 0,C 180,E1 -24988.668,E2 -24988.668} C_VEL
LIN {X 0,Y 146.44,Z 428.246,A -85,B 0,C 180,E1 -24991.394,E2 -24991.394} C_VEL
LIN {X 0,Y 140.286,Z 417.705,A -85,B 0,C 180,E1 -24994.573,E2 -24994.573} C_VEL
LIN {X 0,Y 136.253,Z 411.15,A -85,B 0,C 180,E1 -24996.879,E2 -24996.879} C_VEL
LIN {X 0,Y 133.84,Z 407.381,A -85,B 0,C 180,E1 -24998.348,E2 -24998.348} C_VEL
LIN {X 0,Y 131.406,Z 403.431,A -85,B 0,C 180,E1 -24999.862,E2 -24999.862} C_VEL
LIN {X 0,Y 129.694,Z 401.133,A -85,B 0,C 180,E1 -25000.925,E2 -25000.925} C_VEL
LIN {X 0,Y 129.088,Z 399.01,A -85,B 0,C 180,E1 -25001.552,E2 -25001.552} C_VEL
LIN {X 0,Y 129.331,Z 398.977,A -85,B 0,C 180,E1 -25007.973,E2 -25007.973} C_VEL
LIN {X 0,Y 129.448,Z 398.959,A -85,B 0,C 180,E1 -25010.627,E2 -25010.627} C_VEL
LIN {X 0,Y 130.055,Z 398.912,A -85,B 0,C 180,E1 -25020.001,E2 -25020.001} C_VEL
LIN {X 0,Y 129.45,Z 398.975,A -85,B 0,C 180,E1 -25029.375,E2 -25029.375} C_VEL
LIN {X 0,Y 129.286,Z 399.004,A -85,B 0,C 180,E1 -25032.56,E2 -25032.56} C_VEL
LIN {X 0,Y 129.07,Z 399.023,A -85,B 0,C 180,E1 -25039.07,E2 -25039.07} C_VEL
LIN {X 0,Y 129.023,Z 399.037,A -85,B 0,C 180,E1 -25042.415,E2 -25042.415} C_VEL
LIN {X 0,Y 128.99,Z 399.041,A -85,B 0,C 180,E1 -25049.366,E2 -25049.366} C_VEL
LIN {X 0,Y 128.947,Z 399.033,A -85,B 0,C 180,E1 -25055.169,E2 -25055.169} C_VEL
LIN {X 0,Y 128.915,Z 399.041,A -85,B 0,C 180,E1 -25060.86,E2 -25060.86} C_VEL
LIN {X 0,Y 128.905,Z 399.049,A -85,B 0,C 180,E1 -25065.136,E2 -25065.136} C_VEL
LIN {X 0,Y 128.927,Z 399.037,A -85,B 0,C 180,E1 -25069.745,E2 -25069.745} C_VEL
LIN {X 0,Y 128.95,Z 399.047,A -85,B 0,C 180,E1 -25074.839,E2 -25074.839} C_VEL
LIN {X 0,Y 129.013,Z 399.036,A -85,B 0,C 180,E1 -25080.647,E2 -25080.647} C_VEL
LIN {X 0,Y 129.009,Z 399.034,A -85,B 0,C 180,E1 -25084.168,E2 -25084.168} C_VEL
LIN {X 0,Y 129.069,Z 399.031,A -85,B 0,C 180,E1 -25087.773,E2 -25087.773} C_VEL
LIN {X 0,Y 129.152,Z 398.984,A -85,B 0,C 180,E1 -25094.217,E2 -25094.217} C_VEL
LIN {X 0,Y 129.345,Z 398.982,A -85,B 0,C 180,E1 -25097.973,E2 -25097.973} C_VEL
LIN {X 0,Y 129.463,Z 398.984,A -85,B 0,C 180,E1 -25100.632,E2 -25100.632} C_VEL
LIN {X 0,Y 130.07,Z 398.909,A -85,B 0,C 180,E1 -25110.005,E2 -25110.005} C_VEL
LIN {X 0,Y 129.915,Z 398.955,A -85,B 0,C 180,E1 -25110.78,E2 -25110.78} C_VEL
LIN {X 0,Y 130.87,Z 401.869,A -85,B 0,C 180,E1 -25111.591,E2 -25111.591} C_VEL
LIN {X 0,Y 132.477,Z 404.066,A -85,B 0,C 180,E1 -25112.57,E2 -25112.57} C_VEL
LIN {X 0,Y 134.529,Z 407.526,A -85,B 0,C 180,E1 -25113.841,E2 -25113.841} C_VEL
LIN {X 0,Y 140.027,Z 416.516,A -85,B 0,C 180,E1 -25117.061,E2 -25117.061} C_VEL
LIN {X 0,Y 148.779,Z 432.415,A -85,B 0,C 180,E1 -25121.63,E2 -25121.63} C_VEL
LIN {X 0,Y 156.33,Z 447.433,A -85,B 0,C 180,E1 -25125.21,E2 -25125.21} C_VEL
LIN {X 0,Y 164.512,Z 465.069,A -85,B 0,C 180,E1 -25128.737,E2 -25128.737} C_VEL
LIN {X 0,Y 166.755,Z 470.012,A -85,B 0,C 180,E1 -25129.647,E2 -25129.647} C_VEL
LIN {X 0,Y 157.746,Z 547.753,A -85,B 0,C 180,E1 -25134.123,E2 -25134.123} C_VEL
LIN {X 0,Y 155.251,Z 563.683,A -85,B 0,C 180,E1 -25135.506,E2 -25135.506} C_VEL
LIN {X 0,Y 152.118,Z 579.67,A -85,B 0,C 180,E1 -25137.417,E2 -25137.417} C_VEL
LIN {X 0,Y 148.65,Z 594.163,A -85,B 0,C 180,E1 -25139.685,E2 -25139.685} C_VEL
LIN {X 0,Y 144.793,Z 608.604,A -85,B 0,C 180,E1 -25142.583,E2 -25142.583} C_VEL
LIN {X 0,Y 140.949,Z 621.642,A -85,B 0,C 180,E1 -25145.877,E2 -25145.877} C_VEL
LIN {X 0,Y 137.188,Z 634,A -85,B 0,C 180,E1 -25149.785,E2 -25149.785} C_VEL
LIN {X 0,Y 134.001,Z 644.43,A -85,B 0,C 180,E1 -25153.849,E2 -25153.849} C_VEL
LIN {X 0,Y 130.952,Z 655,A -85,B 0,C 180,E1 -25158.925,E2 -25158.925} C_VEL
LIN {X 0,Y 128.684,Z 664.055,A -85,B 0,C 180,E1 -25164.32,E2 -25164.32} C_VEL
LIN {X 0,Y 127.394,Z 670.908,A -85,B 0,C 180,E1 -25169.315,E2 -25169.315} C_VEL
LIN {X 0,Y 126.39,Z 677.6,A -85,B 0,C 180,E1 -25175.351,E2 -25175.351} C_VEL
LIN {X 0,Y 126.003,Z 682.918,A -85,B 0,C 180,E1 -25181.49,E2 -25181.49} C_VEL
LIN {X 0,Y 126.326,Z 686.696,A -85,B 0,C 180,E1 -25187.141,E2 -25187.141} C_VEL
LIN {X 0,Y 127.906,Z 689.984,A -85,B 0,C 180,E1 -25193.69,E2 -25193.69} C_VEL
LIN {X 0,Y 130.647,Z 692.109,A -85,B 0,C 180,E1 -25199.999,E2 -25199.999} C_VEL
LIN {X 0,Y 134.849,Z 693.136,A -85,B 0,C 180,E1 -25205.982,E2 -25205.982} C_VEL
LIN {X 0,Y 140.454,Z 693.196,A -85,B 0,C 180,E1 -25211.545,E2 -25211.545} C_VEL
LIN {X 0,Y 147.346,Z 692.27,A -85,B 0,C 180,E1 -25216.629,E2 -25216.629} C_VEL
LIN {X 0,Y 155.406,Z 690.318,A -85,B 0,C 180,E1 -25221.209,E2 -25221.209} C_VEL
LIN {X 0,Y 164.553,Z 687.366,A -85,B 0,C 180,E1 -25225.283,E2 -25225.283} C_VEL
LIN {X 0,Y 174.711,Z 683.366,A -85,B 0,C 180,E1 -25228.862,E2 -25228.862} C_VEL
LIN {X 0,Y 188.46,Z 676.719,A -85,B 0,C 180,E1 -25232.733,E2 -25232.733} C_VEL
LIN {X 0,Y 196.122,Z 672.419,A -85,B 0,C 180,E1 -25234.488,E2 -25234.488} C_VEL
LIN {X 0,Y 196.706,Z 672.077,A -85,B 0,C 180,E1 -25234.735,E2 -25234.735} C_VEL
LIN {X 0,Y 185.46,Z 678.749,A -85,B 0,C 180,E1 -25237.265,E2 -25237.265} C_VEL
LIN {X 0,Y 174.774,Z 684.319,A -85,B 0,C 180,E1 -25240.175,E2 -25240.175} C_VEL
LIN {X 0,Y 164.79,Z 688.83,A -85,B 0,C 180,E1 -25243.525,E2 -25243.525} C_VEL
LIN {X 0,Y 155.749,Z 692.435,A -85,B 0,C 180,E1 -25247.397,E2 -25247.397} C_VEL
LIN {X 0,Y 146.447,Z 695.412,A -85,B 0,C 180,E1 -25252.654,E2 -25252.654} C_VEL
LIN {X 0,Y 137.724,Z 697.384,A -85,B 0,C 180,E1 -25259.312,E2 -25259.312} C_VEL
LIN {X 0,Y 133.374,Z 697.741,A -85,B 0,C 180,E1 -25264.006,E2 -25264.006} C_VEL
LIN {X 0,Y 131.073,Z 697.689,A -85,B 0,C 180,E1 -25266.361,E2 -25266.361} C_VEL
LIN {X 0,Y 126.065,Z 696.981,A -85,B 0,C 180,E1 -25270.162,E2 -25270.162} C_VEL
LIN {X 0,Y 122.351,Z 696.013,A -85,B 0,C 180,E1 -25273.379,E2 -25273.379} C_VEL
LIN {X 0,Y 120.581,Z 695.104,A -85,B 0,C 180,E1 -25276.011,E2 -25276.011} C_VEL
LIN {X 0,Y 120.305,Z 694.761,A -85,B 0,C 180,E1 -25276.928,E2 -25276.928} C_VEL
LIN {X 0,Y 119.739,Z 692.185,A -85,B 0,C 180,E1 -25283.254,E2 -25283.254} C_VEL
LIN {X 0,Y 119.923,Z 689.865,A -85,B 0,C 180,E1 -25287.549,E2 -25287.549} C_VEL
LIN {X 0,Y 120.047,Z 686.992,A -85,B 0,C 180,E1 -25291.672,E2 -25291.672} C_VEL
LIN {X 0,Y 120.038,Z 682.575,A -85,B 0,C 180,E1 -25296.719,E2 -25296.719} C_VEL
LIN {X 0,Y 120.736,Z 675.216,A -85,B 0,C 180,E1 -25303.459,E2 -25303.459} C_VEL
LIN {X 0,Y 122.226,Z 667.187,A -85,B 0,C 180,E1 -25309.301,E2 -25309.301} C_VEL
LIN {X 0,Y 124.408,Z 659.141,A -85,B 0,C 180,E1 -25314.092,E2 -25314.092} C_VEL
LIN {X 0,Y 127.33,Z 649.504,A -85,B 0,C 180,E1 -25318.783,E2 -25318.783} C_VEL
LIN {X 0,Y 130.925,Z 637.777,A -85,B 0,C 180,E1 -25323.376,E2 -25323.376} C_VEL
LIN {X 0,Y 134.956,Z 625.3,A -85,B 0,C 180,E1 -25327.251,E2 -25327.251} C_VEL
LIN {X 0,Y 138.961,Z 611.865,A -85,B 0,C 180,E1 -25330.562,E2 -25330.562} C_VEL
LIN {X 0,Y 143.099,Z 596.854,A -85,B 0,C 180,E1 -25333.432,E2 -25333.432} C_VEL
LIN {X 0,Y 146.719,Z 581.536,A -85,B 0,C 180,E1 -25335.68,E2 -25335.68} C_VEL
LIN {X 0,Y 149.68,Z 566.688,A -85,B 0,C 180,E1 -25337.31,E2 -25337.31} C_VEL
LIN {X 0,Y 152.087,Z 551.265,A -85,B 0,C 180,E1 -25338.538,E2 -25338.538} C_VEL
LIN {X 0,Y 160.524,Z 478.619,A -85,B 0,C 180,E1 -25342.889,E2 -25342.889} C_VEL
LIN {X 0,Y 153.889,Z 460.546,A -85,B 0,C 180,E1 -25346.094,E2 -25346.094} C_VEL
LIN {X 0,Y 146.431,Z 441.793,A -85,B 0,C 180,E1 -25350.025,E2 -25350.025} C_VEL
LIN {X 0,Y 139.48,Z 428.716,A -85,B 0,C 180,E1 -25353.663,E2 -25353.663} C_VEL
LIN {X 0,Y 132.388,Z 416.646,A -85,B 0,C 180,E1 -25357.83,E2 -25357.83} C_VEL
LIN {X 0,Y 127.22,Z 408.627,A -85,B 0,C 180,E1 -25361.104,E2 -25361.104} C_VEL
LIN {X 0,Y 125.154,Z 405.195,A -85,B 0,C 180,E1 -25362.581,E2 -25362.581} C_VEL
LIN {X 0,Y 122.82,Z 402.238,A -85,B 0,C 180,E1 -25364.229,E2 -25364.229} C_VEL
LIN {X 0,Y 122.089,Z 399.904,A -85,B 0,C 180,E1 -25364.988,E2 -25364.988} C_VEL
LIN {X 0,Y 122.377,Z 399.836,A -85,B 0,C 180,E1 -25370.08,E2 -25370.08} C_VEL
LIN {X 0,Y 122.545,Z 399.837,A -85,B 0,C 180,E1 -25376.713,E2 -25376.713} C_VEL
LIN {X 0,Y 123.008,Z 399.789,A -85,B 0,C 180,E1 -25380.001,E2 -25380.001} C_VEL
LIN {X 0,Y 122.375,Z 399.864,A -85,B 0,C 180,E1 -25386.883,E2 -25386.883} C_VEL
LIN {X 0,Y 122.275,Z 399.875,A -85,B 0,C 180,E1 -25392.31,E2 -25392.31} C_VEL
LIN {X 0,Y 122.048,Z 399.894,A -85,B 0,C 180,E1 -25396.734,E2 -25396.734} C_VEL
LIN {X 0,Y 121.968,Z 399.915,A -85,B 0,C 180,E1 -25402.802,E2 -25402.802} C_VEL
LIN {X 0,Y 121.906,Z 399.925,A -85,B 0,C 180,E1 -25410.155,E2 -25410.155} C_VEL
LIN {X 0,Y 121.872,Z 399.92,A -85,B 0,C 180,E1 -25416.173,E2 -25416.173} C_VEL
LIN {X 0,Y 121.838,Z 399.918,A -85,B 0,C 180,E1 -25421.428,E2 -25421.428} C_VEL
LIN {X 0,Y 121.856,Z 399.925,A -85,B 0,C 180,E1 -25428.572,E2 -25428.572} C_VEL
LIN {X 0,Y 121.902,Z 399.925,A -85,B 0,C 180,E1 -25434.8,E2 -25434.8} C_VEL
LIN {X 0,Y 121.922,Z 399.913,A -85,B 0,C 180,E1 -25439.845,E2 -25439.845} C_VEL
LIN {X 0,Y 121.961,Z 399.908,A -85,B 0,C 180,E1 -25446.216,E2 -25446.216} C_VEL
LIN {X 0,Y 121.992,Z 399.914,A -85,B 0,C 180,E1 -25449.783,E2 -25449.783} C_VEL
LIN {X 0,Y 122.188,Z 399.857,A -85,B 0,C 180,E1 -25456.704,E2 -25456.704} C_VEL
LIN {X 0,Y 122.392,Z 399.866,A -85,B 0,C 180,E1 -25460.085,E2 -25460.085} C_VEL
LIN {X 0,Y 122.619,Z 399.82,A -85,B 0,C 180,E1 -25467.13,E2 -25467.13} C_VEL
LIN {X 0,Y 123.694,Z 402.606,A -85,B 0,C 180,E1 -25468.173,E2 -25468.173} C_VEL
LIN {X 0,Y 125.839,Z 404.905,A -85,B 0,C 180,E1 -25469.605,E2 -25469.605} C_VEL
LIN {X 0,Y 127.658,Z 408.261,A -85,B 0,C 180,E1 -25470.936,E2 -25470.936} C_VEL
LIN {X 0,Y 135.403,Z 420.934,A -85,B 0,C 180,E1 -25475.788,E2 -25475.788} C_VEL
LIN {X 0,Y 143.988,Z 436.988,A -85,B 0,C 180,E1 -25480.586,E2 -25480.586} C_VEL
LIN {X 0,Y 151.008,Z 451.03,A -85,B 0,C 180,E1 -25484.093,E2 -25484.093} C_VEL
LIN {X 0,Y 160.539,Z 471.914,A -85,B 0,C 180,E1 -25488.373,E2 -25488.373} C_VEL
LIN {X 0,Y 152.715,Z 538.016,A -85,B 0,C 180,E1 -25492.267,E2 -25492.267} C_VEL
LIN {X 0,Y 150.232,Z 555.7,A -85,B 0,C 180,E1 -25493.562,E2 -25493.562} C_VEL
LIN {X 0,Y 147.256,Z 572.133,A -85,B 0,C 180,E1 -25495.325,E2 -25495.325} C_VEL
LIN {X 0,Y 143.684,Z 587.738,A -85,B 0,C 180,E1 -25497.556,E2 -25497.556} C_VEL
LIN {X 0,Y 139.715,Z 602.826,A -85,B 0,C 180,E1 -25500.376,E2 -25500.376} C_VEL
LIN {X 0,Y 135.426,Z 617.356,A -85,B 0,C 180,E1 -25503.866,E2 -25503.866} C_VEL
LIN {X 0,Y 131.343,Z 630.46,A -85,B 0,C 180,E1 -25507.882,E2 -25507.882} C_VEL
LIN {X 0,Y 127.524,Z 642.444,A -85,B 0,C 180,E1 -25512.513,E2 -25512.513} C_VEL
LIN {X 0,Y 124.535,Z 652.491,A -85,B 0,C 180,E1 -25517.373,E2 -25517.373} C_VEL
LIN {X 0,Y 122.145,Z 661.303,A -85,B 0,C 180,E1 -25522.629,E2 -25522.629} C_VEL
LIN {X 0,Y 120.509,Z 669.134,A -85,B 0,C 180,E1 -25528.339,E2 -25528.339} C_VEL
LIN {X 0,Y 119.543,Z 675.319,A -85,B 0,C 180,E1 -25533.836,E2 -25533.836} C_VEL
LIN {X 0,Y 118.996,Z 680.302,A -85,B 0,C 180,E1 -25539.244,E2 -25539.244} C_VEL
LIN {X 0,Y 119.038,Z 684.25,A -85,B 0,C 180,E1 -25544.592,E2 -25544.592} C_VEL
LIN {X 0,Y 119.676,Z 687.384,A -85,B 0,C 180,E1 -25549.852,E2 -25549.852} C_VEL
LIN {X 0,Y 121.805,Z 690.503,A -85,B 0,C 180,E1 -25556.691,E2 -25556.691} C_VEL
LIN {X 0,Y 125.299,Z 692.528,A -85,B 0,C 180,E1 -25563.214,E2 -25563.214} C_VEL
LIN {X 0,Y 130.27,Z 693.473,A -85,B 0,C 180,E1 -25569.313,E2 -25569.313} C_VEL
LIN {X 0,Y 136.692,Z 693.456,A -85,B 0,C 180,E1 -25574.896,E2 -25574.896} C_VEL
LIN {X 0,Y 144.364,Z 692.512,A -85,B 0,C 180,E1 -25579.923,E2 -25579.923} C_VEL
LIN {X 0,Y 155.63,Z 689.893,A -85,B 0,C 180,E1 -25585.415,E2 -25585.415} C_VEL
LIN {X 0,Y 168.393,Z 685.676,A -85,B 0,C 180,E1 -25590.054,E2 -25590.054} C_VEL
LIN {X 0,Y 179.601,Z 681.097,A -85,B 0,C 180,E1 -25593.218,E2 -25593.218} C_VEL
LIN {X 0,Y 184.998,Z 678.554,A -85,B 0,C 180,E1 -25594.549,E2 -25594.549} C_VEL
LIN {X 0,Y 182.887,Z 679.648,A -85,B 0,C 180,E1 -25595.176,E2 -25595.176} C_VEL
LIN {X 0,Y 170.353,Z 685.59,A -85,B 0,C 180,E1 -25598.38,E2 -25598.38} C_VEL
LIN {X 0,Y 160.035,Z 689.813,A -85,B 0,C 180,E1 -25601.702,E2 -25601.702} C_VEL
LIN {X 0,Y 150.624,Z 693.009,A -85,B 0,C 180,E1 -25605.577,E2 -25605.577} C_VEL
LIN {X 0,Y 142.235,Z 695.386,A -85,B 0,C 180,E1 -25610.028,E2 -25610.028} C_VEL
LIN {X 0,Y 134.922,Z 696.851,A -85,B 0,C 180,E1 -25615.036,E2 -25615.036} C_VEL
LIN {X 0,Y 127.572,Z 697.443,A -85,B 0,C 180,E1 -25621.816,E2 -25621.816} C_VEL
LIN {X 0,Y 124.228,Z 697.144,A -85,B 0,C 180,E1 -25626.666,E2 -25626.666} C_VEL
LIN {X 0,Y 121.297,Z 695.896,A -85,B 0,C 180,E1 -25633.155,E2 -25633.155} C_VEL
LIN {X 0,Y 120.305,Z 694.761,A -85,B 0,C 180,E1 -25636.928,E2 -25636.928} C_VEL
LIN {X 0,Y 119.274,Z 693.676,A -85,B 0,C 180,E1 -25639.655,E2 -25639.655} C_VEL
LIN {X 0,Y 117.59,Z 692.229,A -85,B 0,C 180,E1 -25642.325,E2 -25642.325} C_VEL
LIN {X 0,Y 114.048,Z 688.597,A -85,B 0,C 180,E1 -25647.724,E2 -25647.724} C_VEL
LIN {X 0,Y 113.04,Z 685.8,A -85,B 0,C 180,E1 -25651.482,E2 -25651.482} C_VEL
LIN {X 0,Y 113.056,Z 681.033,A -85,B 0,C 180,E1 -25657.137,E2 -25657.137} C_VEL
LIN {X 0,Y 113.874,Z 673.329,A -85,B 0,C 180,E1 -25664.287,E2 -25664.287} C_VEL
LIN {X 0,Y 115.593,Z 664.958,A -85,B 0,C 180,E1 -25670.457,E2 -25670.457} C_VEL
LIN {X 0,Y 118.272,Z 655.407,A -85,B 0,C 180,E1 -25676.122,E2 -25676.122} C_VEL
LIN {X 0,Y 121.747,Z 644.516,A -85,B 0,C 180,E1 -25681.295,E2 -25681.295} C_VEL
LIN {X 0,Y 125.795,Z 632.226,A -85,B 0,C 180,E1 -25685.911,E2 -25685.911} C_VEL
LIN {X 0,Y 130.171,Z 618.641,A -85,B 0,C 180,E1 -25689.87,E2 -25689.87} C_VEL
LIN {X 0,Y 134.148,Z 605.319,A -85,B 0,C 180,E1 -25692.92,E2 -25692.92} C_VEL
LIN {X 0,Y 138.286,Z 590.056,A -85,B 0,C 180,E1 -25695.61,E2 -25695.61} C_VEL
LIN {X 0,Y 141.859,Z 574.191,A -85,B 0,C 180,E1 -25697.727,E2 -25697.727} C_VEL
LIN {X 0,Y 144.838,Z 557.917,A -85,B 0,C 180,E1 -25699.296,E2 -25699.296} C_VEL
LIN {X 0,Y 148.435,Z 529.077,A -85,B 0,C 180,E1 -25701.231,E2 -25701.231} C_VEL
LIN {X 0,Y 154.394,Z 480.309,A -85,B 0,C 180,E1 -25704.197,E2 -25704.197} C_VEL
LIN {X 0,Y 147.04,Z 460.221,A -85,B 0,C 180,E1 -25708.013,E2 -25708.013} C_VEL
LIN {X 0,Y 140.976,Z 444.875,A -85,B 0,C 180,E1 -25711.428,E2 -25711.428} C_VEL
LIN {X 0,Y 133.552,Z 430.971,A -85,B 0,C 180,E1 -25715.635,E2 -25715.635} C_VEL
LIN {X 0,Y 127.782,Z 421.185,A -85,B 0,C 180,E1 -25719.213,E2 -25719.213} C_VEL
LIN {X 0,Y 122.973,Z 413.553,A -85,B 0,C 180,E1 -25722.527,E2 -25722.527} C_VEL
LIN {X 0,Y 120.71,Z 409.897,A -85,B 0,C 180,E1 -25724.271,E2 -25724.271} C_VEL
LIN {X 0,Y 118.52,Z 406.623,A -85,B 0,C 180,E1 -25725.952,E2 -25725.952} C_VEL
LIN {X 0,Y 117.9,Z 405.544,A -85,B 0,C 180,E1 -25726.469,E2 -25726.469} C_VEL
LIN {X 0,Y 116.005,Z 403.159,A -85,B 0,C 180,E1 -25727.973,E2 -25727.973} C_VEL
LIN {X 0,Y 115.257,Z 400.722,A -85,B 0,C 180,E1 -25728.924,E2 -25728.924} C_VEL
LIN {X 0,Y 115.334,Z 400.736,A -85,B 0,C 180,E1 -25733.001,E2 -25733.001} C_VEL
LIN {X 0,Y 115.96,Z 400.667,A -85,B 0,C 180,E1 -25740.001,E2 -25740.001} C_VEL
LIN {X 0,Y 115.335,Z 400.744,A -85,B 0,C 180,E1 -25747.001,E2 -25747.001} C_VEL
LIN {X 0,Y 115.192,Z 400.758,A -85,B 0,C 180,E1 -25752.559,E2 -25752.559} C_VEL
LIN {X 0,Y 114.953,Z 400.776,A -85,B 0,C 180,E1 -25757.801,E2 -25757.801} C_VEL
LIN {X 0,Y 114.883,Z 400.793,A -85,B 0,C 180,E1 -25763.432,E2 -25763.432} C_VEL
LIN {X 0,Y 114.838,Z 400.803,A -85,B 0,C 180,E1 -25771.053,E2 -25771.053} C_VEL
LIN {X 0,Y 114.767,Z 400.812,A -85,B 0,C 180,E1 -25777.763,E2 -25777.763} C_VEL
LIN {X 0,Y 114.762,Z 400.797,A -85,B 0,C 180,E1 -25782.712,E2 -25782.712} C_VEL
LIN {X 0,Y 114.779,Z 400.81,A -85,B 0,C 180,E1 -25787.667,E2 -25787.667} C_VEL
LIN {X 0,Y 114.777,Z 400.805,A -85,B 0,C 180,E1 -25792.753,E2 -25792.753} C_VEL
LIN {X 0,Y 114.85,Z 400.79,A -85,B 0,C 180,E1 -25798.95,E2 -25798.95} C_VEL
LIN {X 0,Y 114.925,Z 400.785,A -85,B 0,C 180,E1 -25806.536,E2 -25806.536} C_VEL
LIN {X 0,Y 114.969,Z 400.763,A -85,B 0,C 180,E1 -25812.209,E2 -25812.209} C_VEL
LIN {X 0,Y 115.306,Z 400.745,A -85,B 0,C 180,E1 -25819.469,E2 -25819.469} C_VEL
LIN {X 0,Y 115.361,Z 400.724,A -85,B 0,C 180,E1 -25823.117,E2 -25823.117} C_VEL
LIN {X 0,Y 116.308,Z 403.429,A -85,B 0,C 180,E1 -25824.153,E2 -25824.153} C_VEL
LIN {X 0,Y 118.43,Z 405.646,A -85,B 0,C 180,E1 -25825.751,E2 -25825.751} C_VEL
LIN {X 0,Y 121.338,Z 409.719,A -85,B 0,C 180,E1 -25827.929,E2 -25827.929} C_VEL
LIN {X 0,Y 122.445,Z 411.417,A -85,B 0,C 180,E1 -25828.77,E2 -25828.77} C_VEL
LIN {X 0,Y 130.025,Z 424.113,A -85,B 0,C 180,E1 -25833.988,E2 -25833.988} C_VEL
LIN {X 0,Y 138.695,Z 440.335,A -85,B 0,C 180,E1 -25839.186,E2 -25839.186} C_VEL
LIN {X 0,Y 146.86,Z 457.116,A -85,B 0,C 180,E1 -25843.475,E2 -25843.475} C_VEL
LIN {X 0,Y 154.407,Z 474.008,A -85,B 0,C 180,E1 -25847.089,E2 -25847.089} C_VEL
LIN {X 0,Y 145.263,Z 547.227,A -85,B 0,C 180,E1 -25851.59,E2 -25851.59} C_VEL
LIN {X 0,Y 142.546,Z 563.588,A -85,B 0,C 180,E1 -25853.086,E2 -25853.086} C_VEL
LIN {X 0,Y 139.21,Z 579.446,A -85,B 0,C 180,E1 -25855.097,E2 -25855.097} C_VEL
LIN {X 0,Y 135.62,Z 593.641,A -85,B 0,C 180,E1 -25857.445,E2 -25857.445} C_VEL
LIN {X 0,Y 131.529,Z 607.996,A -85,B 0,C 180,E1 -25860.5,E2 -25860.5} C_VEL
LIN {X 0,Y 127.357,Z 621.331,A -85,B 0,C 180,E1 -25864.13,E2 -25864.13} C_VEL
LIN {X 0,Y 123.302,Z 633.783,A -85,B 0,C 180,E1 -25868.436,E2 -25868.436} C_VEL
LIN {X 0,Y 119.317,Z 646.061,A -85,B 0,C 180,E1 -25873.816,E2 -25873.816} C_VEL
LIN {X 0,Y 116.282,Z 656.297,A -85,B 0,C 180,E1 -25879.478,E2 -25879.478} C_VEL
LIN {X 0,Y 114.211,Z 664.885,A -85,B 0,C 180,E1 -25885.367,E2 -25885.367} C_VEL
LIN {X 0,Y 113.044,Z 671.129,A -85,B 0,C 180,E1 -25890.513,E2 -25890.513} C_VEL
LIN {X 0,Y 112.209,Z 676.532,A -85,B 0,C 180,E1 -25895.975,E2 -25895.975} C_VEL
LIN {X 0,Y 111.906,Z 681.271,A -85,B 0,C 180,E1 -25901.698,E2 -25901.698} C_VEL
LIN {X 0,Y 112.466,Z 686.142,A -85,B 0,C 180,E1 -25909.194,E2 -25909.194} C_VEL
LIN {X 0,Y 114.525,Z 689.649,A -85,B 0,C 180,E1 -25916.481,E2 -25916.481} C_VEL
LIN {X 0,Y 118.004,Z 692.073,A -85,B 0,C 180,E1 -25923.413,E2 -25923.413} C_VEL
LIN {X 0,Y 123.058,Z 693.496,A -85,B 0,C 180,E1 -25929.864,E2 -25929.864} C_VEL
LIN {X 0,Y 129.64,Z 693.881,A -85,B 0,C 180,E1 -25935.726,E2 -25935.726} C_VEL
LIN {X 0,Y 137.541,Z 693.359,A -85,B 0,C 180,E1 -25940.957,E2 -25940.957} C_VEL
LIN {X 0,Y 146.623,Z 691.883,A -85,B 0,C 180,E1 -25945.555,E2 -25945.555} C_VEL
LIN {X 0,Y 156.753,Z 689.381,A -85,B 0,C 180,E1 -25949.549,E2 -25949.549} C_VEL
LIN {X 0,Y 167.799,Z 685.914,A -85,B 0,C 180,E1 -25952.989,E2 -25952.989} C_VEL
LIN {X 0,Y 173.633,Z 683.756,A -85,B 0,C 180,E1 -25954.517,E2 -25954.517} C_VEL
LIN {X 0,Y 160.733,Z 688.855,A -85,B 0,C 180,E1 -25958.085,E2 -25958.085} C_VEL
LIN {X 0,Y 150.419,Z 692.214,A -85,B 0,C 180,E1 -25961.615,E2 -25961.615} C_VEL
LIN {X 0,Y 141.105,Z 694.712,A -85,B 0,C 180,E1 -25965.784,E2 -25965.784} C_VEL
LIN {X 0,Y 129.146,Z 696.823,A -85,B 0,C 180,E1 -25973.224,E2 -25973.224} C_VEL
LIN {X 0,Y 121.07,Z 697.091,A -85,B 0,C 180,E1 -25980.543,E2 -25980.543} C_VEL
LIN {X 0,Y 115.867,Z 695.997,A -85,B 0,C 180,E1 -25988.653,E2 -25988.653} C_VEL
LIN {X 0,Y 113.335,Z 693.707,A -85,B 0,C 180,E1 -25996.514,E2 -25996.514} C_VEL
LIN {X 0,Y 112.836,Z 689.844,A -85,B 0,C 180,E1 -26005.238,E2 -26005.238} C_VEL
LIN {X 0,Y 113.073,Z 686.923,A -85,B 0,C 180,E1 -26009.995,E2 -26009.995} C_VEL
LIN {X 0,Y 113.04,Z 685.8,A -85,B 0,C 180,E1 -26011.482,E2 -26011.482} C_VEL
LIN {X 0,Y 112.415,Z 683.529,A -85,B 0,C 180,E1 -26014.213,E2 -26014.213} C_VEL
LIN {X 0,Y 110.944,Z 680.943,A -85,B 0,C 180,E1 -26016.842,E2 -26016.842} C_VEL
LIN {X 0,Y 107.686,Z 675.02,A -85,B 0,C 180,E1 -26022.075,E2 -26022.075} C_VEL
LIN {X 0,Y 107.04,Z 671.843,A -85,B 0,C 180,E1 -26024.769,E2 -26024.769} C_VEL
LIN {X 0,Y 107.121,Z 670.74,A -85,B 0,C 180,E1 -26025.67,E2 -26025.67} C_VEL
LIN {X 0,Y 109.377,Z 661.172,A -85,B 0,C 180,E1 -26032.67,E2 -26032.67} C_VEL
LIN {X 0,Y 112.621,Z 650.61,A -85,B 0,C 180,E1 -26038.759,E2 -26038.759} C_VEL
LIN {X 0,Y 116.356,Z 639.196,A -85,B 0,C 180,E1 -26043.96,E2 -26043.96} C_VEL
LIN {X 0,Y 120.924,Z 625.995,A -85,B 0,C 180,E1 -26048.659,E2 -26048.659} C_VEL
LIN {X 0,Y 125.215,Z 612.712,A -85,B 0,C 180,E1 -26052.333,E2 -26052.333} C_VEL
LIN {X 0,Y 129.52,Z 598.34,A -85,B 0,C 180,E1 -26055.406,E2 -26055.406} C_VEL
LIN {X 0,Y 133.386,Z 583.639,A -85,B 0,C 180,E1 -26057.804,E2 -26057.804} C_VEL
LIN {X 0,Y 136.867,Z 567.26,A -85,B 0,C 180,E1 -26059.795,E2 -26059.795} C_VEL
LIN {X 0,Y 139.55,Z 551.272,A -85,B 0,C 180,E1 -26061.165,E2 -26061.165} C_VEL
LIN {X 0,Y 148.291,Z 481.984,A -85,B 0,C 180,E1 -26065.578,E2 -26065.578} C_VEL
LIN {X 0,Y 140.622,Z 460.767,A -85,B 0,C 180,E1 -26069.893,E2 -26069.893} C_VEL
LIN {X 0,Y 135.633,Z 448.316,A -85,B 0,C 180,E1 -26072.863,E2 -26072.863} C_VEL
LIN {X 0,Y 128.565,Z 434.732,A -85,B 0,C 180,E1 -26077.195,E2 -26077.195} C_VEL
LIN {X 0,Y 122.015,Z 423.513,A -85,B 0,C 180,E1 -26081.614,E2 -26081.614} C_VEL
LIN {X 0,Y 116.769,Z 415.219,A -85,B 0,C 180,E1 -26085.626,E2 -26085.626} C_VEL
LIN {X 0,Y 113.971,Z 410.875,A -85,B 0,C 180,E1 -26087.981,E2 -26087.981} C_VEL
LIN {X 0,Y 111.968,Z 407.71,A -85,B 0,C 180,E1 -26089.833,E2 -26089.833} C_VEL
LIN {X 0,Y 111.338,Z 406.62,A -85,B 0,C 180,E1 -26090.463,E2 -26090.463} C_VEL
LIN {X 0,Y 109.272,Z 404.45,A -85,B 0,C 180,E1 -26092.378,E2 -26092.378} C_VEL
LIN {X 0,Y 108.359,Z 402.092,A -85,B 0,C 180,E1 -26093.484,E2 -26093.484} C_VEL
LIN {X 0,Y 108.298,Z 401.619,A -85,B 0,C 180,E1 -26093.714,E2 -26093.714} C_VEL
LIN {X 0,Y 108.885,Z 401.548,A -85,B 0,C 180,E1 -26100.001,E2 -26100.001} C_VEL
LIN {X 0,Y 108.275,Z 401.622,A -85,B 0,C 180,E1 -26107.46,E2 -26107.46} C_VEL
LIN {X 0,Y 108.126,Z 401.64,A -85,B 0,C 180,E1 -26112.874,E2 -26112.874} C_VEL
LIN {X 0,Y 107.849,Z 401.664,A -85,B 0,C 180,E1 -26119.017,E2 -26119.017} C_VEL
LIN {X 0,Y 107.792,Z 401.671,A -85,B 0,C 180,E1 -26124.12,E2 -26124.12} C_VEL
LIN {X 0,Y 107.764,Z 401.677,A -85,B 0,C 180,E1 -26132.036,E2 -26132.036} C_VEL
LIN {X 0,Y 107.674,Z 401.696,A -85,B 0,C 180,E1 -26138.45,E2 -26138.45} C_VEL
LIN {X 0,Y 107.66,Z 401.697,A -85,B 0,C 180,E1 -26145.897,E2 -26145.897} C_VEL
LIN {X 0,Y 107.676,Z 401.681,A -85,B 0,C 180,E1 -26151.56,E2 -26151.56} C_VEL
LIN {X 0,Y 107.786,Z 401.669,A -85,B 0,C 180,E1 -26158.566,E2 -26158.566} C_VEL
LIN {X 0,Y 107.888,Z 401.663,A -85,B 0,C 180,E1 -26166.999,E2 -26166.999} C_VEL
LIN {X 0,Y 107.97,Z 401.618,A -85,B 0,C 180,E1 -26174.914,E2 -26174.914} C_VEL
LIN {X 0,Y 108.202,Z 401.61,A -85,B 0,C 180,E1 -26178.146,E2 -26178.146} C_VEL
LIN {X 0,Y 109.133,Z 404.241,A -85,B 0,C 180,E1 -26179.395,E2 -26179.395} C_VEL
LIN {X 0,Y 111.128,Z 406.491,A -85,B 0,C 180,E1 -26181.252,E2 -26181.252} C_VEL
LIN {X 0,Y 111.858,Z 407.135,A -85,B 0,C 180,E1 -26181.879,E2 -26181.879} C_VEL
LIN {X 0,Y 113.68,Z 410.276,A -85,B 0,C 180,E1 -26183.625,E2 -26183.625} C_VEL
LIN {X 0,Y 115.496,Z 412.302,A -85,B 0,C 180,E1 -26185.075,E2 -26185.075} C_VEL
LIN {X 0,Y 118.518,Z 416.715,A -85,B 0,C 180,E1 -26187.454,E2 -26187.454} C_VEL
LIN {X 0,Y 126.381,Z 430.156,A -85,B 0,C 180,E1 -26193.193,E2 -26193.193} C_VEL
LIN {X 0,Y 134.055,Z 445.006,A -85,B 0,C 180,E1 -26198.049,E2 -26198.049} C_VEL
LIN {X 0,Y 142.077,Z 461.833,A -85,B 0,C 180,E1 -26202.522,E2 -26202.522} C_VEL
LIN {X 0,Y 148.299,Z 476.263,A -85,B 0,C 180,E1 -26205.723,E2 -26205.723} C_VEL
LIN {X 0,Y 139.042,Z 547.431,A -85,B 0,C 180,E1 -26210.204,E2 -26210.204} C_VEL
LIN {X 0,Y 136.216,Z 563.918,A -85,B 0,C 180,E1 -26211.764,E2 -26211.764} C_VEL
LIN {X 0,Y 132.631,Z 580.168,A -85,B 0,C 180,E1 -26213.925,E2 -26213.925} C_VEL
LIN {X 0,Y 128.428,Z 595.869,A -85,B 0,C 180,E1 -26216.702,E2 -26216.702} C_VEL
LIN {X 0,Y 124.244,Z 609.735,A -85,B 0,C 180,E1 -26219.892,E2 -26219.892} C_VEL
LIN {X 0,Y 119.732,Z 623.606,A -85,B 0,C 180,E1 -26223.991,E2 -26223.991} C_VEL
LIN {X 0,Y 115.656,Z 635.63,A -85,B 0,C 180,E1 -26228.52,E2 -26228.52} C_VEL
LIN {X 0,Y 111.898,Z 647.055,A -85,B 0,C 180,E1 -26233.947,E2 -26233.947} C_VEL
LIN {X 0,Y 108.954,Z 656.924,A -85,B 0,C 180,E1 -26239.83,E2 -26239.83} C_VEL
LIN {X 0,Y 106.936,Z 665.262,A -85,B 0,C 180,E1 -26246.037,E2 -26246.037} C_VEL
LIN {X 0,Y 105.672,Z 672.103,A -85,B 0,C 180,E1 -26252.253,E2 -26252.253} C_VEL
LIN {X 0,Y 104.918,Z 678.703,A -85,B 0,C 180,E1 -26259.7,E2 -26259.7} C_VEL
LIN {X 0,Y 105.099,Z 683.423,A -85,B 0,C 180,E1 -26266.464,E2 -26266.464} C_VEL
LIN {X 0,Y 106.223,Z 687.073,A -85,B 0,C 180,E1 -26272.993,E2 -26272.993} C_VEL
LIN {X 0,Y 108.751,Z 690.175,A -85,B 0,C 180,E1 -26279.999,E2 -26279.999} C_VEL
LIN {X 0,Y 113.455,Z 692.59,A -85,B 0,C 180,E1 -26287.604,E2 -26287.604} C_VEL
LIN {X 0,Y 119.05,Z 693.836,A -85,B 0,C 180,E1 -26293.658,E2 -26293.658} C_VEL
LIN {X 0,Y 126.932,Z 694.187,A -85,B 0,C 180,E1 -26299.724,E2 -26299.724} C_VEL
LIN {X 0,Y 135.258,Z 693.636,A -85,B 0,C 180,E1 -26304.561,E2 -26304.561} C_VEL
LIN {X 0,Y 145.146,Z 692.154,A -85,B 0,C 180,E1 -26308.959,E2 -26308.959} C_VEL
LIN {X 0,Y 156.006,Z 689.667,A -85,B 0,C 180,E1 -26312.723,E2 -26312.723} C_VEL
LIN {X 0,Y 162.042,Z 687.96,A -85,B 0,C 180,E1 -26314.501,E2 -26314.501} C_VEL
LIN {X 0,Y 151.033,Z 691.461,A -85,B 0,C 180,E1 -26317.71,E2 -26317.71} C_VEL
LIN {X 0,Y 140.853,Z 694.024,A -85,B 0,C 180,E1 -26321.539,E2 -26321.539} C_VEL
LIN {X 0,Y 131.622,Z 695.792,A -85,B 0,C 180,E1 -26326.036,E2 -26326.036} C_VEL
LIN {X 0,Y 123.519,Z 696.697,A -85,B 0,C 180,E1 -26331.248,E2 -26331.248} C_VEL
LIN {X 0,Y 114.57,Z 696.594,A -85,B 0,C 180,E1 -26339.18,E2 -26339.18} C_VEL
LIN {X 0,Y 109.269,Z 695.226,A -85,B 0,C 180,E1 -26347.294,E2 -26347.294} C_VEL
LIN {X 0,Y 106.662,Z 693.086,A -85,B 0,C 180,E1 -26354.713,E2 -26354.713} C_VEL
LIN {X 0,Y 105.8,Z 689.903,A -85,B 0,C 180,E1 -26362.36,E2 -26362.36} C_VEL
LIN {X 0,Y 106.025,Z 686.757,A -85,B 0,C 180,E1 -26368.095,E2 -26368.095} C_VEL
LIN {X 0,Y 106.058,Z 684.111,A -85,B 0,C 180,E1 -26371.893,E2 -26371.893} C_VEL
LIN {X 0,Y 106.082,Z 679.273,A -85,B 0,C 180,E1 -26377.608,E2 -26377.608} C_VEL
LIN {X 0,Y 106.842,Z 672.402,A -85,B 0,C 180,E1 -26384.275,E2 -26384.275} C_VEL
LIN {X 0,Y 107.121,Z 670.74,A -85,B 0,C 180,E1 -26385.67,E2 -26385.67} C_VEL
LIN {X 0,Y 107.067,Z 667.402,A -85,B 0,C 180,E1 -26388.273,E2 -26388.273} C_VEL
LIN {X 0,Y 105.628,Z 661.365,A -85,B 0,C 180,E1 -26392.444,E2 -26392.444} C_VEL
LIN {X 0,Y 104.656,Z 654.927,A -85,B 0,C 180,E1 -26396.536,E2 -26396.536} C_VEL
LIN {X 0,Y 105.343,Z 650.833,A -85,B 0,C 180,E1 -26398.888,E2 -26398.888} C_VEL
LIN {X 0,Y 109.092,Z 639.765,A -85,B 0,C 180,E1 -26404.305,E2 -26404.305} C_VEL
LIN {X 0,Y 113.74,Z 626.71,A -85,B 0,C 180,E1 -26409.29,E2 -26409.29} C_VEL
LIN {X 0,Y 118.157,Z 613.643,A -85,B 0,C 180,E1 -26413.151,E2 -26413.151} C_VEL
LIN {X 0,Y 122.627,Z 599.199,A -85,B 0,C 180,E1 -26416.453,E2 -26416.453} C_VEL
LIN {X 0,Y 126.781,Z 584.154,A -85,B 0,C 180,E1 -26419.043,E2 -26419.043} C_VEL
LIN {X 0,Y 130.38,Z 568.202,A -85,B 0,C 180,E1 -26421.091,E2 -26421.091} C_VEL
LIN {X 0,Y 133.269,Z 551.844,A -85,B 0,C 180,E1 -26422.583,E2 -26422.583} C_VEL
LIN {X 0,Y 142.249,Z 483.783,A -85,B 0,C 180,E1 -26427.081,E2 -26427.081} C_VEL
LIN {X 0,Y 134.798,Z 462.799,A -85,B 0,C 180,E1 -26431.553,E2 -26431.553} C_VEL
LIN {X 0,Y 130.615,Z 452.194,A -85,B 0,C 180,E1 -26434.275,E2 -26434.275} C_VEL
LIN {X 0,Y 123.75,Z 438.777,A -85,B 0,C 180,E1 -26438.732,E2 -26438.732} C_VEL
LIN {X 0,Y 117.653,Z 428.093,A -85,B 0,C 180,E1 -26443.239,E2 -26443.239} C_VEL
LIN {X 0,Y 112.894,Z 420.457,A -85,B 0,C 180,E1 -26447.073,E2 -26447.073} C_VEL
LIN {X 0,Y 110.202,Z 416.168,A -85,B 0,C 180,E1 -26449.552,E2 -26449.552} C_VEL
LIN {X 0,Y 107.869,Z 412.439,A -85,B 0,C 180,E1 -26451.925,E2 -26451.925} C_VEL
LIN {X 0,Y 105.622,Z 409.59,A -85,B 0,C 180,E1 -26454.147,E2 -26454.147} C_VEL
LIN {X 0,Y 104.887,Z 407.796,A -85,B 0,C 180,E1 -26455.1,E2 -26455.1} C_VEL
LIN {X 0,Y 102.816,Z 405.857,A -85,B 0,C 180,E1 -26457.308,E2 -26457.308} C_VEL
LIN {X 0,Y 101.772,Z 403.235,A -85,B 0,C 180,E1 -26458.888,E2 -26458.888} C_VEL
LIN {X 0,Y 101.704,Z 402.439,A -85,B 0,C 180,E1 -26459.259,E2 -26459.259} C_VEL
LIN {X 0,Y 101.813,Z 402.429,A -85,B 0,C 180,E1 -26460.001,E2 -26460.001} C_VEL
LIN {X 0,Y 101.209,Z 402.498,A -85,B 0,C 180,E1 -26467.984,E2 -26467.984} C_VEL
LIN {X 0,Y 101.039,Z 402.524,A -85,B 0,C 180,E1 -26473.173,E2 -26473.173} C_VEL
LIN {X 0,Y 100.763,Z 402.555,A -85,B 0,C 180,E1 -26480.412,E2 -26480.412} C_VEL
LIN {X 0,Y 100.707,Z 402.549,A -85,B 0,C 180,E1 -26484.891,E2 -26484.891} C_VEL
LIN {X 0,Y 100.676,Z 402.552,A -85,B 0,C 180,E1 -26493.114,E2 -26493.114} C_VEL
LIN {X 0,Y 100.623,Z 402.57,A -85,B 0,C 180,E1 -26499.81,E2 -26499.81} C_VEL
LIN {X 0,Y 100.631,Z 402.572,A -85,B 0,C 180,E1 -26505.711,E2 -26505.711} C_VEL
LIN {X 0,Y 100.614,Z 402.559,A -85,B 0,C 180,E1 -26511.057,E2 -26511.057} C_VEL
LIN {X 0,Y 100.683,Z 402.558,A -85,B 0,C 180,E1 -26516.894,E2 -26516.894} C_VEL
LIN {X 0,Y 100.738,Z 402.55,A -85,B 0,C 180,E1 -26525.09,E2 -26525.09} C_VEL
LIN {X 0,Y 100.834,Z 402.703,A -85,B 0,C 180,E1 -26531.925,E2 -26531.925} C_VEL
LIN {X 0,Y 101.65,Z 405.047,A -85,B 0,C 180,E1 -26533.306,E2 -26533.306} C_VEL
LIN {X 0,Y 103.834,Z 407.342,A -85,B 0,C 180,E1 -26535.823,E2 -26535.823} C_VEL
LIN {X 0,Y 104.981,Z 408.235,A -85,B 0,C 180,E1 -26536.975,E2 -26536.975} C_VEL
LIN {X 0,Y 106.905,Z 411.478,A -85,B 0,C 180,E1 -26539.111,E2 -26539.111} C_VEL
LIN {X 0,Y 108.697,Z 413.421,A -85,B 0,C 180,E1 -26540.76,E2 -26540.76} C_VEL
LIN {X 0,Y 110.962,Z 416.789,A -85,B 0,C 180,E1 -26542.955,E2 -26542.955} C_VEL
LIN {X 0,Y 112.485,Z 418.858,A -85,B 0,C 180,E1 -26544.292,E2 -26544.292} C_VEL
LIN {X 0,Y 114.947,Z 422.485,A -85,B 0,C 180,E1 -26546.349,E2 -26546.349} C_VEL
LIN {X 0,Y 122.413,Z 435.692,A -85,B 0,C 180,E1 -26552.122,E2 -26552.122} C_VEL
LIN {X 0,Y 129.568,Z 449.991,A -85,B 0,C 180,E1 -26556.923,E2 -26556.923} C_VEL
LIN {X 0,Y 136.914,Z 465.719,A -85,B 0,C 180,E1 -26561.326,E2 -26561.326} C_VEL
LIN {X 0,Y 142.266,Z 478.069,A -85,B 0,C 180,E1 -26564.203,E2 -26564.203} C_VEL
LIN {X 0,Y 132.86,Z 547.423,A -85,B 0,C 180,E1 -26568.741,E2 -26568.741} C_VEL
LIN {X 0,Y 129.823,Z 564.376,A -85,B 0,C 180,E1 -26570.408,E2 -26570.408} C_VEL
LIN {X 0,Y 126.386,Z 579.446,A -85,B 0,C 180,E1 -26572.454,E2 -26572.454} C_VEL
LIN {X 0,Y 122.288,Z 594.473,A -85,B 0,C 180,E1 -26575.152,E2 -26575.152} C_VEL
LIN {X 0,Y 117.832,Z 608.807,A -85,B 0,C 180,E1 -26578.505,E2 -26578.505} C_VEL
LIN {X 0,Y 113.004,Z 623.211,A -85,B 0,C 180,E1 -26582.904,E2 -26582.904} C_VEL
LIN {X 0,Y 108.751,Z 635.302,A -85,B 0,C 180,E1 -26587.658,E2 -26587.658} C_VEL
LIN {X 0,Y 105.261,Z 645.507,A -85,B 0,C 180,E1 -26592.738,E2 -26592.738} C_VEL
LIN {X 0,Y 101.981,Z 656.039,A -85,B 0,C 180,E1 -26599.302,E2 -26599.302} C_VEL
LIN {X 0,Y 99.921,Z 664.361,A -85,B 0,C 180,E1 -26605.757,E2 -26605.757} C_VEL
LIN {X 0,Y 98.598,Z 671.392,A -85,B 0,C 180,E1 -26612.397,E2 -26612.397} C_VEL
LIN {X 0,Y 97.935,Z 676.998,A -85,B 0,C 180,E1 -26618.972,E2 -26618.972} C_VEL
LIN {X 0,Y 98.171,Z 682.886,A -85,B 0,C 180,E1 -26627.597,E2 -26627.597} C_VEL
LIN {X 0,Y 99.981,Z 687.372,A -85,B 0,C 180,E1 -26635.968,E2 -26635.968} C_VEL
LIN {X 0,Y 103.454,Z 690.641,A -85,B 0,C 180,E1 -26643.894,E2 -26643.894} C_VEL
LIN {X 0,Y 108.706,Z 692.854,A -85,B 0,C 180,E1 -26651.183,E2 -26651.183} C_VEL
LIN {X 0,Y 115.63,Z 694.16,A -85,B 0,C 180,E1 -26657.691,E2 -26657.691} C_VEL
LIN {X 0,Y 124.001,Z 694.497,A -85,B 0,C 180,E1 -26663.373,E2 -26663.373} C_VEL
LIN {X 0,Y 133.587,Z 693.926,A -85,B 0,C 180,E1 -26668.26,E2 -26668.26} C_VEL
LIN {X 0,Y 144.236,Z 692.468,A -85,B 0,C 180,E1 -26672.41,E2 -26672.41} C_VEL
LIN {X 0,Y 149.918,Z 691.333,A -85,B 0,C 180,E1 -26674.231,E2 -26674.231} C_VEL
LIN {X 0,Y 146.817,Z 692.144,A -85,B 0,C 180,E1 -26675.528,E2 -26675.528} C_VEL
LIN {X 0,Y 136.259,Z 694.421,A -85,B 0,C 180,E1 -26679.309,E2 -26679.309} C_VEL
LIN {X 0,Y 126.585,Z 695.86,A -85,B 0,C 180,E1 -26683.794,E2 -26683.794} C_VEL
LIN {X 0,Y 118.037,Z 696.517,A -85,B 0,C 180,E1 -26689.078,E2 -26689.078} C_VEL
LIN {X 0,Y 110.628,Z 696.297,A -85,B 0,C 180,E1 -26695.121,E2 -26695.121} C_VEL
LIN {X 0,Y 104.945,Z 695.268,A -85,B 0,C 180,E1 -26702.039,E2 -26702.039} C_VEL
LIN {X 0,Y 101.104,Z 693.334,A -85,B 0,C 180,E1 -26709.656,E2 -26709.656} C_VEL
LIN {X 0,Y 99.131,Z 690.441,A -85,B 0,C 180,E1 -26717.714,E2 -26717.714} C_VEL
LIN {X 0,Y 98.994,Z 686.524,A -85,B 0,C 180,E1 -26725.923,E2 -26725.923} C_VEL
LIN {X 0,Y 99.159,Z 684.005,A -85,B 0,C 180,E1 -26729.994,E2 -26729.994} C_VEL
LIN {X 0,Y 99.092,Z 678.628,A -85,B 0,C 180,E1 -26736.821,E2 -26736.821} C_VEL
LIN {X 0,Y 99.843,Z 671.347,A -85,B 0,C 180,E1 -26744.256,E2 -26744.256} C_VEL
LIN {X 0,Y 101.657,Z 662.768,A -85,B 0,C 180,E1 -26751.275,E2 -26751.275} C_VEL
LIN {X 0,Y 104.28,Z 654.06,A -85,B 0,C 180,E1 -26757.053,E2 -26757.053} C_VEL
LIN {X 0,Y 105.343,Z 650.833,A -85,B 0,C 180,E1 -26758.888,E2 -26758.888} C_VEL
LIN {X 0,Y 106.119,Z 646.699,A -85,B 0,C 180,E1 -26761.116,E2 -26761.116} C_VEL
LIN {X 0,Y 105.805,Z 639.461,A -85,B 0,C 180,E1 -26764.748,E2 -26764.748} C_VEL
LIN {X 0,Y 105.669,Z 631.856,A -85,B 0,C 180,E1 -26768.242,E2 -26768.242} C_VEL
LIN {X 0,Y 106.703,Z 627.096,A -85,B 0,C 180,E1 -26770.102,E2 -26770.102} C_VEL
LIN {X 0,Y 111.595,Z 613.148,A -85,B 0,C 180,E1 -26774.469,E2 -26774.469} C_VEL
LIN {X 0,Y 116.164,Z 598.855,A -85,B 0,C 180,E1 -26777.858,E2 -26777.858} C_VEL
LIN {X 0,Y 120.544,Z 583.512,A -85,B 0,C 180,E1 -26780.571,E2 -26780.571} C_VEL
LIN {X 0,Y 124.412,Z 566.734,A -85,B 0,C 180,E1 -26782.755,E2 -26782.755} C_VEL
LIN {X 0,Y 127.259,Z 550.971,A -85,B 0,C 180,E1 -26784.198,E2 -26784.198} C_VEL
LIN {X 0,Y 136.238,Z 485.399,A -85,B 0,C 180,E1 -26788.654,E2 -26788.654} C_VEL
LIN {X 0,Y 128.467,Z 463.037,A -85,B 0,C 180,E1 -26793.812,E2 -26793.812} C_VEL
LIN {X 0,Y 125.37,Z 455.508,A -85,B 0,C 180,E1 -26795.911,E2 -26795.911} C_VEL
LIN {X 0,Y 119.283,Z 443.391,A -85,B 0,C 180,E1 -26800.185,E2 -26800.185} C_VEL
LIN {X 0,Y 113.523,Z 433.051,A -85,B 0,C 180,E1 -26804.713,E2 -26804.713} C_VEL
LIN {X 0,Y 108.988,Z 425.517,A -85,B 0,C 180,E1 -26808.729,E2 -26808.729} C_VEL
LIN {X 0,Y 106.084,Z 420.754,A -85,B 0,C 180,E1 -26811.668,E2 -26811.668} C_VEL
LIN {X 0,Y 104.381,Z 418.081,A -85,B 0,C 180,E1 -26813.444,E2 -26813.444} C_VEL
LIN {X 0,Y 102.157,Z 414.837,A -85,B 0,C 180,E1 -26815.937,E2 -26815.937} C_VEL
LIN {X 0,Y 101.5,Z 413.669,A -85,B 0,C 180,E1 -26816.776,E2 -26816.776} C_VEL
LIN {X 0,Y 99.36,Z 410.876,A -85,B 0,C 180,E1 -26819.495,E2 -26819.495} C_VEL
LIN {X 0,Y 98.616,Z 408.865,A -85,B 0,C 180,E1 -26820.792,E2 -26820.792} C_VEL
LIN {X 0,Y 95.76,Z 406.915,A -85,B 0,C 180,E1 -26824.474,E2 -26824.474} C_VEL
LIN {X 0,Y 94.455,Z 404.686,A -85,B 0,C 180,E1 -26826.812,E2 -26826.812} C_VEL
LIN {X 0,Y 94.176,Z 403.375,A -85,B 0,C 180,E1 -26827.775,E2 -26827.775} C_VEL
LIN {X 0,Y 93.947,Z 403.408,A -85,B 0,C 180,E1 -26833.498,E2 -26833.498} C_VEL
LIN {X 0,Y 93.633,Z 403.446,A -85,B 0,C 180,E1 -26842.044,E2 -26842.044} C_VEL
LIN {X 0,Y 93.577,Z 403.437,A -85,B 0,C 180,E1 -26846.785,E2 -26846.785} C_VEL
LIN {X 0,Y 93.573,Z 403.434,A -85,B 0,C 180,E1 -26854.304,E2 -26854.304} C_VEL
LIN {X 0,Y 93.517,Z 403.441,A -85,B 0,C 180,E1 -26862.562,E2 -26862.562} C_VEL
LIN {X 0,Y 93.523,Z 403.449,A -85,B 0,C 180,E1 -26868.72,E2 -26868.72} C_VEL
LIN {X 0,Y 93.579,Z 403.451,A -85,B 0,C 180,E1 -26875.705,E2 -26875.705} C_VEL
LIN {X 0,Y 93.64,Z 403.65,A -85,B 0,C 180,E1 -26883.603,E2 -26883.603} C_VEL
LIN {X 0,Y 94.77,Z 406.417,A -85,B 0,C 180,E1 -26886.053,E2 -26886.053} C_VEL
LIN {X 0,Y 96.737,Z 408.397,A -85,B 0,C 180,E1 -26888.995,E2 -26888.995} C_VEL
LIN {X 0,Y 97.971,Z 409.317,A -85,B 0,C 180,E1 -26890.567,E2 -26890.567} C_VEL
LIN {X 0,Y 99.925,Z 412.585,A -85,B 0,C 180,E1 -26893.378,E2 -26893.378} C_VEL
LIN {X 0,Y 102.057,Z 414.669,A -85,B 0,C 180,E1 -26895.833,E2 -26895.833} C_VEL
LIN {X 0,Y 104.429,Z 418.159,A -85,B 0,C 180,E1 -26898.512,E2 -26898.512} C_VEL
LIN {X 0,Y 105.546,Z 419.613,A -85,B 0,C 180,E1 -26899.638,E2 -26899.638} C_VEL
LIN {X 0,Y 109.088,Z 424.639,A -85,B 0,C 180,E1 -26903.064,E2 -26903.064} C_VEL
LIN {X 0,Y 111.454,Z 428.37,A -85,B 0,C 180,E1 -26905.221,E2 -26905.221} C_VEL
LIN {X 0,Y 118.206,Z 440.683,A -85,B 0,C 180,E1 -26910.767,E2 -26910.767} C_VEL
LIN {X 0,Y 124.756,Z 454.251,A -85,B 0,C 180,E1 -26915.564,E2 -26915.564} C_VEL
LIN {X 0,Y 130.873,Z 467.534,A -85,B 0,C 180,E1 -26919.472,E2 -26919.472} C_VEL
LIN {X 0,Y 136.145,Z 480.01,A -85,B 0,C 180,E1 -26922.607,E2 -26922.607} C_VEL
LIN {X 0,Y 126.735,Z 547.428,A -85,B 0,C 180,E1 -26927.149,E2 -26927.149} C_VEL
LIN {X 0,Y 123.751,Z 563.782,A -85,B 0,C 180,E1 -26928.783,E2 -26928.783} C_VEL
LIN {X 0,Y 119.982,Z 579.724,A -85,B 0,C 180,E1 -26931.003,E2 -26931.003} C_VEL
LIN {X 0,Y 115.415,Z 595.752,A -85,B 0,C 180,E1 -26934.018,E2 -26934.018} C_VEL
LIN {X 0,Y 110.898,Z 609.615,A -85,B 0,C 180,E1 -26937.47,E2 -26937.47} C_VEL
LIN {X 0,Y 105.993,Z 623.623,A -85,B 0,C 180,E1 -26942.042,E2 -26942.042} C_VEL
LIN {X 0,Y 101.504,Z 635.886,A -85,B 0,C 180,E1 -26947.228,E2 -26947.228} C_VEL
LIN {X 0,Y 97.316,Z 647.873,A -85,B 0,C 180,E1 -26953.763,E2 -26953.763} C_VEL
LIN {X 0,Y 94.261,Z 657.77,A -85,B 0,C 180,E1 -26960.671,E2 -26960.671} C_VEL
LIN {X 0,Y 92.377,Z 665.962,A -85,B 0,C 180,E1 -26967.82,E2 -26967.82} C_VEL
LIN {X 0,Y 91.289,Z 672.581,A -85,B 0,C 180,E1 -26974.948,E2 -26974.948} C_VEL
LIN {X 0,Y 90.856,Z 677.944,A -85,B 0,C 180,E1 -26981.975,E2 -26981.975} C_VEL
LIN {X 0,Y 91.292,Z 682.349,A -85,B 0,C 180,E1 -26988.902,E2 -26988.902} C_VEL
LIN {X 0,Y 92.726,Z 685.876,A -85,B 0,C 180,E1 -26995.652,E2 -26995.652} C_VEL
LIN {X 0,Y 96.189,Z 689.606,A -85,B 0,C 180,E1 -27004.189,E2 -27004.189} C_VEL
LIN {X 0,Y 101.571,Z 692.254,A -85,B 0,C 180,E1 -27011.979,E2 -27011.979} C_VEL
LIN {X 0,Y 108.675,Z 693.956,A -85,B 0,C 180,E1 -27018.865,E2 -27018.865} C_VEL
LIN {X 0,Y 117.317,Z 694.78,A -85,B 0,C 180,E1 -27024.792,E2 -27024.792} C_VEL
LIN {X 0,Y 127.166,Z 694.634,A -85,B 0,C 180,E1 -27029.827,E2 -27029.827} C_VEL
LIN {X 0,Y 138.09,Z 693.646,A -85,B 0,C 180,E1 -27034.044,E2 -27034.044} C_VEL
LIN {X 0,Y 137.239,Z 693.858,A -85,B 0,C 180,E1 -27034.973,E2 -27034.973} C_VEL
LIN {X 0,Y 121.76,Z 695.862,A -85,B 0,C 180,E1 -27041.372,E2 -27041.372} C_VEL
LIN {X 0,Y 112.749,Z 696.21,A -85,B 0,C 180,E1 -27046.705,E2 -27046.705} C_VEL
LIN {X 0,Y 101.937,Z 695.296,A -85,B 0,C 180,E1 -27055.824,E2 -27055.824} C_VEL
LIN {X 0,Y 96.323,Z 693.483,A -85,B 0,C 180,E1 -27064.031,E2 -27064.031} C_VEL
LIN {X 0,Y 93.154,Z 690.896,A -85,B 0,C 180,E1 -27072.429,E2 -27072.429} C_VEL
LIN {X 0,Y 91.976,Z 686.208,A -85,B 0,C 180,E1 -27083.38,E2 -27083.38} C_VEL
LIN {X 0,Y 92.162,Z 683.745,A -85,B 0,C 180,E1 -27087.808,E2 -27087.808} C_VEL
LIN {X 0,Y 92.118,Z 680.82,A -85,B 0,C 180,E1 -27092.18,E2 -27092.18} C_VEL
LIN {X 0,Y 92.161,Z 675.537,A -85,B 0,C 180,E1 -27098.766,E2 -27098.766} C_VEL
LIN {X 0,Y 93.215,Z 667.976,A -85,B 0,C 180,E1 -27106.416,E2 -27106.416} C_VEL
LIN {X 0,Y 95.571,Z 658.781,A -85,B 0,C 180,E1 -27113.85,E2 -27113.85} C_VEL
LIN {X 0,Y 98.998,Z 648.374,A -85,B 0,C 180,E1 -27120.482,E2 -27120.482} C_VEL
LIN {X 0,Y 102.904,Z 637.209,A -85,B 0,C 180,E1 -27126.082,E2 -27126.082} C_VEL
LIN {X 0,Y 106.703,Z 627.096,A -85,B 0,C 180,E1 -27130.102,E2 -27130.102} C_VEL
LIN {X 0,Y 107.762,Z 622.306,A -85,B 0,C 180,E1 -27131.861,E2 -27131.861} C_VEL
LIN {X 0,Y 107.861,Z 614.089,A -85,B 0,C 180,E1 -27134.817,E2 -27134.817} C_VEL
LIN {X 0,Y 108.026,Z 605.664,A -85,B 0,C 180,E1 -27137.593,E2 -27137.593} C_VEL
LIN {X 0,Y 109.129,Z 600.394,A -85,B 0,C 180,E1 -27138.952,E2 -27138.952} C_VEL
LIN {X 0,Y 113.576,Z 585.821,A -85,B 0,C 180,E1 -27141.773,E2 -27141.773} C_VEL
LIN {X 0,Y 117.678,Z 569.65,A -85,B 0,C 180,E1 -27144.084,E2 -27144.084} C_VEL
LIN {X 0,Y 120.883,Z 553.01,A -85,B 0,C 180,E1 -27145.748,E2 -27145.748} C_VEL
LIN {X 0,Y 130.243,Z 486.987,A -85,B 0,C 180,E1 -27150.379,E2 -27150.379} C_VEL
LIN {X 0,Y 123.368,Z 466.721,A -85,B 0,C 180,E1 -27155.305,E2 -27155.305} C_VEL
LIN {X 0,Y 120.559,Z 459.658,A -85,B 0,C 180,E1 -27157.382,E2 -27157.382} C_VEL
LIN {X 0,Y 114.805,Z 447.818,A -85,B 0,C 180,E1 -27161.81,E2 -27161.81} C_VEL
LIN {X 0,Y 109.329,Z 437.823,A -85,B 0,C 180,E1 -27166.407,E2 -27166.407} C_VEL
LIN {X 0,Y 105.35,Z 430.804,A -85,B 0,C 180,E1 -27170.337,E2 -27170.337} C_VEL
LIN {X 0,Y 101.424,Z 424.202,A -85,B 0,C 180,E1 -27174.584,E2 -27174.584} C_VEL
LIN {X 0,Y 99.059,Z 420.685,A -85,B 0,C 180,E1 -27177.46,E2 -27177.46} C_VEL
LIN {X 0,Y 97.805,Z 418.843,A -85,B 0,C 180,E1 -27179.145,E2 -27179.145} C_VEL
LIN {X 0,Y 95.91,Z 415.582,A -85,B 0,C 180,E1 -27181.97,E2 -27181.97} C_VEL
LIN {X 0,Y 92.652,Z 412.376,A -85,B 0,C 180,E1 -27186.879,E2 -27186.879} C_VEL
LIN {X 0,Y 91.517,Z 409.98,A -85,B 0,C 180,E1 -27189.382,E2 -27189.382} C_VEL
LIN {X 0,Y 88.342,Z 408.005,A -85,B 0,C 180,E1 -27195.874,E2 -27195.874} C_VEL
LIN {X 0,Y 86.78,Z 405.365,A -85,B 0,C 180,E1 -27201.374,E2 -27201.374} C_VEL
LIN {X 0,Y 86.554,Z 404.319,A -85,B 0,C 180,E1 -27203.32,E2 -27203.32} C_VEL
LIN {X 0,Y 86.444,Z 404.341,A -85,B 0,C 180,E1 -27209.198,E2 -27209.198} C_VEL
LIN {X 0,Y 86.492,Z 404.319,A -85,B 0,C 180,E1 -27215.666,E2 -27215.666} C_VEL
LIN {X 0,Y 86.441,Z 404.322,A -85,B 0,C 180,E1 -27222.979,E2 -27222.979} C_VEL
LIN {X 0,Y 86.496,Z 404.514,A -85,B 0,C 180,E1 -27228.868,E2 -27228.868} C_VEL
LIN {X 0,Y 87.135,Z 406.635,A -85,B 0,C 180,E1 -27232.399,E2 -27232.399} C_VEL
LIN {X 0,Y 90.096,Z 409.653,A -85,B 0,C 180,E1 -27240.032,E2 -27240.032} C_VEL
LIN {X 0,Y 91.311,Z 410.462,A -85,B 0,C 180,E1 -27242.349,E2 -27242.349} C_VEL
LIN {X 0,Y 93.021,Z 413.685,A -85,B 0,C 180,E1 -27245.934,E2 -27245.934} C_VEL
LIN {X 0,Y 95.239,Z 415.656,A -85,B 0,C 180,E1 -27249.226,E2 -27249.226} C_VEL
LIN {X 0,Y 97.519,Z 419.112,A -85,B 0,C 180,E1 -27252.509,E2 -27252.509} C_VEL
LIN {X 0,Y 99.11,Z 420.815,A -85,B 0,C 180,E1 -27254.506,E2 -27254.506} C_VEL
LIN {X 0,Y 101.61,Z 424.408,A -85,B 0,C 180,E1 -27257.509,E2 -27257.509} C_VEL
LIN {X 0,Y 106.655,Z 431.738,A -85,B 0,C 180,E1 -27262.654,E2 -27262.654} C_VEL
LIN {X 0,Y 113.728,Z 445.084,A -85,B 0,C 180,E1 -27269.133,E2 -27269.133} C_VEL
LIN {X 0,Y 119.967,Z 458.392,A -85,B 0,C 180,E1 -27274.063,E2 -27274.063} C_VEL
LIN {X 0,Y 126.064,Z 472.066,A -85,B 0,C 180,E1 -27278.254,E2 -27278.254} C_VEL
LIN {X 0,Y 130.252,Z 482.249,A -85,B 0,C 180,E1 -27280.94,E2 -27280.94} C_VEL
LIN {X 0,Y 120.736,Z 547.297,A -85,B 0,C 180,E1 -27285.396,E2 -27285.396} C_VEL
LIN {X 0,Y 117.638,Z 563.653,A -85,B 0,C 180,E1 -27287.08,E2 -27287.08} C_VEL
LIN {X 0,Y 113.638,Z 579.823,A -85,B 0,C 180,E1 -27289.41,E2 -27289.41} C_VEL
LIN {X 0,Y 109.044,Z 595.317,A -85,B 0,C 180,E1 -27292.441,E2 -27292.441} C_VEL
LIN {X 0,Y 104.504,Z 608.807,A -85,B 0,C 180,E1 -27295.907,E2 -27295.907} C_VEL
LIN {X 0,Y 99.432,Z 622.821,A -85,B 0,C 180,E1 -27300.638,E2 -27300.638} C_VEL
LIN {X 0,Y 95.082,Z 634.214,A -85,B 0,C 180,E1 -27305.601,E2 -27305.601} C_VEL
LIN {X 0,Y 90.605,Z 646.494,A -85,B 0,C 180,E1 -27312.531,E2 -27312.531} C_VEL
LIN {X 0,Y 87.352,Z 656.556,A -85,B 0,C 180,E1 -27319.934,E2 -27319.934} C_VEL
LIN {X 0,Y 85.375,Z 664.925,A -85,B 0,C 180,E1 -27327.65,E2 -27327.65} C_VEL
LIN {X 0,Y 84.257,Z 671.749,A -85,B 0,C 180,E1 -27335.35,E2 -27335.35} C_VEL
LIN {X 0,Y 83.89,Z 677.193,A -85,B 0,C 180,E1 -27342.948,E2 -27342.948} C_VEL
LIN {X 0,Y 84.96,Z 683.081,A -85,B 0,C 180,E1 -27353.105,E2 -27353.105} C_VEL
LIN {X 0,Y 86.956,Z 686.414,A -85,B 0,C 180,E1 -27359.999,E2 -27359.999} C_VEL
LIN {X 0,Y 93.134,Z 690.838,A -85,B 0,C 180,E1 -27371.158,E2 -27371.158} C_VEL
LIN {X 0,Y 101.799,Z 693.55,A -85,B 0,C 180,E1 -27380.192,E2 -27380.192} C_VEL
LIN {X 0,Y 110.704,Z 694.797,A -85,B 0,C 180,E1 -27386.383,E2 -27386.383} C_VEL
LIN {X 0,Y 120.852,Z 695.13,A -85,B 0,C 180,E1 -27391.558,E2 -27391.558} C_VEL
LIN {X 0,Y 127.734,Z 694.894,A -85,B 0,C 180,E1 -27394.373,E2 -27394.373} C_VEL
LIN {X 0,Y 117.175,Z 695.752,A -85,B 0,C 180,E1 -27398.758,E2 -27398.758} C_VEL
LIN {X 0,Y 103.326,Z 695.591,A -85,B 0,C 180,E1 -27407.135,E2 -27407.135} C_VEL
LIN {X 0,Y 95.651,Z 694.417,A -85,B 0,C 180,E1 -27413.991,E2 -27413.991} C_VEL
LIN {X 0,Y 90.01,Z 692.486,A -85,B 0,C 180,E1 -27422.057,E2 -27422.057} C_VEL
LIN {X 0,Y 86.498,Z 689.614,A -85,B 0,C 180,E1 -27431.027,E2 -27431.027} C_VEL
LIN {X 0,Y 85.08,Z 684.864,A -85,B 0,C 180,E1 -27442.41,E2 -27442.41} C_VEL
LIN {X 0,Y 85.272,Z 682.085,A -85,B 0,C 180,E1 -27447.631,E2 -27447.631} C_VEL
LIN {X 0,Y 85.173,Z 678.995,A -85,B 0,C 180,E1 -27452.357,E2 -27452.357} C_VEL
LIN {X 0,Y 85.367,Z 672.436,A -85,B 0,C 180,E1 -27460.668,E2 -27460.668} C_VEL
LIN {X 0,Y 86.728,Z 664.311,A -85,B 0,C 180,E1 -27468.906,E2 -27468.906} C_VEL
LIN {X 0,Y 89.638,Z 654.466,A -85,B 0,C 180,E1 -27476.789,E2 -27476.789} C_VEL
LIN {X 0,Y 93.644,Z 643.246,A -85,B 0,C 180,E1 -27483.729,E2 -27483.729} C_VEL
LIN {X 0,Y 98.111,Z 631.201,A -85,B 0,C 180,E1 -27489.467,E2 -27489.467} C_VEL
LIN {X 0,Y 102.645,Z 619.203,A -85,B 0,C 180,E1 -27493.879,E2 -27493.879} C_VEL
LIN {X 0,Y 107.709,Z 604.839,A -85,B 0,C 180,E1 -27497.912,E2 -27497.912} C_VEL
LIN {X 0,Y 109.129,Z 600.394,A -85,B 0,C 180,E1 -27498.952,E2 -27498.952} C_VEL
LIN {X 0,Y 110.187,Z 595.117,A -85,B 0,C 180,E1 -27500.233,E2 -27500.233} C_VEL
LIN {X 0,Y 109.999,Z 579.059,A -85,B 0,C 180,E1 -27504.274,E2 -27504.274} C_VEL
LIN {X 0,Y 110.568,Z 573.46,A -85,B 0,C 180,E1 -27505.319,E2 -27505.319} C_VEL
LIN {X 0,Y 110.995,Z 571.561,A -85,B 0,C 180,E1 -27505.587,E2 -27505.587} C_VEL
LIN {X 0,Y 114.488,Z 555.314,A -85,B 0,C 180,E1 -27507.356,E2 -27507.356} C_VEL
LIN {X 0,Y 124.408,Z 488.777,A -85,B 0,C 180,E1 -27512.222,E2 -27512.222} C_VEL
LIN {X 0,Y 117.538,Z 468.16,A -85,B 0,C 180,E1 -27517.572,E2 -27517.572} C_VEL
LIN {X 0,Y 114.661,Z 461.22,A -85,B 0,C 180,E1 -27519.917,E2 -27519.917} C_VEL
LIN {X 0,Y 109.108,Z 449.838,A -85,B 0,C 180,E1 -27524.554,E2 -27524.554} C_VEL
LIN {X 0,Y 103.347,Z 438.992,A -85,B 0,C 180,E1 -27530.23,E2 -27530.23} C_VEL
LIN {X 0,Y 98.254,Z 430.014,A -85,B 0,C 180,E1 -27536.092,E2 -27536.092} C_VEL
LIN {X 0,Y 95.84,Z 426.061,A -85,B 0,C 180,E1 -27539.405,E2 -27539.405} C_VEL
LIN {X 0,Y 93.228,Z 421.932,A -85,B 0,C 180,E1 -27543.31,E2 -27543.31} C_VEL
LIN {X 0,Y 90.157,Z 418.475,A -85,B 0,C 180,E1 -27548.519,E2 -27548.519} C_VEL
LIN {X 0,Y 89.369,Z 416.694,A -85,B 0,C 180,E1 -27550.465,E2 -27550.465} C_VEL
LIN {X 0,Y 86.115,Z 414.241,A -85,B 0,C 180,E1 -27557.87,E2 -27557.87} C_VEL
LIN {X 0,Y 84.924,Z 411.595,A -85,B 0,C 180,E1 -27563.279,E2 -27563.279} C_VEL
LIN {X 0,Y 84.665,Z 411.167,A -85,B 0,C 180,E1 -27564.524,E2 -27564.524} C_VEL
LIN {X 0,Y 83.381,Z 410.69,A -85,B 0,C 180,E1 -27576.16,E2 -27576.16} C_VEL
LIN {X 0,Y 84.702,Z 411.244,A -85,B 0,C 180,E1 -27587.647,E2 -27587.647} C_VEL
LIN {X 0,Y 85.465,Z 413.536,A -85,B 0,C 180,E1 -27591.848,E2 -27591.848} C_VEL
LIN {X 0,Y 88.57,Z 416.643,A -85,B 0,C 180,E1 -27600.089,E2 -27600.089} C_VEL
LIN {X 0,Y 89.112,Z 417.093,A -85,B 0,C 180,E1 -27601.146,E2 -27601.146} C_VEL
LIN {X 0,Y 90.76,Z 420.187,A -85,B 0,C 180,E1 -27604.853,E2 -27604.853} C_VEL
LIN {X 0,Y 92.71,Z 422.152,A -85,B 0,C 180,E1 -27608.037,E2 -27608.037} C_VEL
LIN {X 0,Y 95.064,Z 425.575,A -85,B 0,C 180,E1 -27611.583,E2 -27611.583} C_VEL
LIN {X 0,Y 96.449,Z 427.293,A -85,B 0,C 180,E1 -27613.419,E2 -27613.419} C_VEL
LIN {X 0,Y 99.717,Z 432.346,A -85,B 0,C 180,E1 -27617.59,E2 -27617.59} C_VEL
LIN {X 0,Y 103.285,Z 437.598,A -85,B 0,C 180,E1 -27621.383,E2 -27621.383} C_VEL
LIN {X 0,Y 109.703,Z 450.35,A -85,B 0,C 180,E1 -27627.752,E2 -27627.752} C_VEL
LIN {X 0,Y 115.73,Z 463.562,A -85,B 0,C 180,E1 -27632.814,E2 -27632.814} C_VEL
LIN {X 0,Y 122.15,Z 478.58,A -85,B 0,C 180,E1 -27637.58,E2 -27637.58} C_VEL
LIN {X 0,Y 124.395,Z 484.124,A -85,B 0,C 180,E1 -27639.096,E2 -27639.096} C_VEL
LIN {X 0,Y 114.644,Z 547.693,A -85,B 0,C 180,E1 -27643.583,E2 -27643.583} C_VEL
LIN {X 0,Y 111.419,Z 564.102,A -85,B 0,C 180,E1 -27645.329,E2 -27645.329} C_VEL
LIN {X 0,Y 107.407,Z 579.781,A -85,B 0,C 180,E1 -27647.657,E2 -27647.657} C_VEL
LIN {X 0,Y 102.486,Z 595.692,A -85,B 0,C 180,E1 -27650.876,E2 -27650.876} C_VEL
LIN {X 0,Y 97.413,Z 610.14,A -85,B 0,C 180,E1 -27654.81,E2 -27654.81} C_VEL
LIN {X 0,Y 92.165,Z 623.98,A -85,B 0,C 180,E1 -27659.84,E2 -27659.84} C_VEL
LIN {X 0,Y 87.002,Z 636.862,A -85,B 0,C 180,E1 -27666.116,E2 -27666.116} C_VEL
LIN {X 0,Y 82.962,Z 647.685,A -85,B 0,C 180,E1 -27673.044,E2 -27673.044} C_VEL
LIN {X 0,Y 80.025,Z 656.797,A -85,B 0,C 180,E1 -27680.451,E2 -27680.451} C_VEL
LIN {X 0,Y 78.135,Z 665.123,A -85,B 0,C 180,E1 -27688.854,E2 -27688.854} C_VEL
LIN {X 0,Y 77.167,Z 671.155,A -85,B 0,C 180,E1 -27696.344,E2 -27696.344} C_VEL
LIN {X 0,Y 77.126,Z 677.967,A -85,B 0,C 180,E1 -27706.83,E2 -27706.83} C_VEL
LIN {X 0,Y 78.972,Z 683.548,A -85,B 0,C 180,E1 -27717.448,E2 -27717.448} C_VEL
LIN {X 0,Y 84.313,Z 688.742,A -85,B 0,C 180,E1 -27729.595,E2 -27729.595} C_VEL
LIN {X 0,Y 90.961,Z 691.796,A -85,B 0,C 180,E1 -27738.001,E2 -27738.001} C_VEL
LIN {X 0,Y 102.924,Z 694.438,A -85,B 0,C 180,E1 -27747.405,E2 -27747.405} C_VEL
LIN {X 0,Y 115.746,Z 695.434,A -85,B 0,C 180,E1 -27753.955,E2 -27753.955} C_VEL
LIN {X 0,Y 114.477,Z 695.533,A -85,B 0,C 180,E1 -27755.238,E2 -27755.238} C_VEL
LIN {X 0,Y 102.857,Z 695.342,A -85,B 0,C 180,E1 -27761.262,E2 -27761.262} C_VEL
LIN {X 0,Y 90.038,Z 693.566,A -85,B 0,C 180,E1 -27771.35,E2 -27771.35} C_VEL
LIN {X 0,Y 83.842,Z 691.332,A -85,B 0,C 180,E1 -27779.797,E2 -27779.797} C_VEL
LIN {X 0,Y 79.893,Z 688.302,A -85,B 0,C 180,E1 -27789.391,E2 -27789.391} C_VEL
LIN {X 0,Y 78.259,Z 683.548,A -85,B 0,C 180,E1 -27801.05,E2 -27801.05} C_VEL
LIN {X 0,Y 78.376,Z 680.326,A -85,B 0,C 180,E1 -27807.423,E2 -27807.423} C_VEL
LIN {X 0,Y 78.242,Z 677.093,A -85,B 0,C 180,E1 -27812.566,E2 -27812.566} C_VEL
LIN {X 0,Y 78.515,Z 670.141,A -85,B 0,C 180,E1 -27821.611,E2 -27821.611} C_VEL
LIN {X 0,Y 80.144,Z 661.623,A -85,B 0,C 180,E1 -27830.526,E2 -27830.526} C_VEL
